LIN {X 0,Y 473.754,Z 554.719,A -85,B 0,C 180,E1 -7288.302,E2 -7288.302} C_VEL
LIN {X 0,Y 473.675,Z 555.595,A -85,B 0,C 180,E1 -7290.002,E2 -7290.002} C_VEL
LIN {X 0,Y 473.755,Z 554.68,A -85,B 0,C 180,E1 -7291.702,E2 -7291.702} C_VEL
LIN {X 0,Y 473.78,Z 553.677,A -85,B 0,C 180,E1 -7292.552,E2 -7292.552} C_VEL
LIN {X 0,Y 473.765,Z 550.247,A -85,B 0,C 180,E1 -7294.255,E2 -7294.255} C_VEL
LIN {X 0,Y 473.855,Z 546.483,A -85,B 0,C 180,E1 -7295.533,E2 -7295.533} C_VEL
LIN {X 0,Y 473.91,Z 541.553,A -85,B 0,C 180,E1 -7296.815,E2 -7296.815} C_VEL
LIN {X 0,Y 474.03,Z 536.5,A -85,B 0,C 180,E1 -7297.883,E2 -7297.883} C_VEL
LIN {X 0,Y 474.244,Z 528.948,A -85,B 0,C 180,E1 -7299.168,E2 -7299.168} C_VEL
LIN {X 0,Y 474.518,Z 521.272,A -85,B 0,C 180,E1 -7300.238,E2 -7300.238} C_VEL
LIN {X 0,Y 474.789,Z 513.997,A -85,B 0,C 180,E1 -7301.095,E2 -7301.095} C_VEL
LIN {X 0,Y 475.091,Z 505.339,A -85,B 0,C 180,E1 -7301.953,E2 -7301.953} C_VEL
LIN {X 0,Y 475.44,Z 496.569,A -85,B 0,C 180,E1 -7302.68,E2 -7302.68} C_VEL
LIN {X 0,Y 475.821,Z 486.805,A -85,B 0,C 180,E1 -7303.344,E2 -7303.344} C_VEL
LIN {X 0,Y 476.16,Z 475.842,A -85,B 0,C 180,E1 -7303.932,E2 -7303.932} C_VEL
LIN {X 0,Y 476.528,Z 464.628,A -85,B 0,C 180,E1 -7304.384,E2 -7304.384} C_VEL
LIN {X 0,Y 476.701,Z 454.582,A -85,B 0,C 180,E1 -7304.679,E2 -7304.679} C_VEL
LIN {X 0,Y 477.021,Z 436.414,A -85,B 0,C 180,E1 -7304.996,E2 -7304.996} C_VEL
LIN {X 0,Y 477.483,Z 358.709,A -85,B 0,C 180,E1 -7306.226,E2 -7306.226} C_VEL
LIN {X 0,Y 475.642,Z 344.411,A -85,B 0,C 180,E1 -7306.547,E2 -7306.547} C_VEL
LIN {X 0,Y 476.419,Z 320.349,A -85,B 0,C 180,E1 -7309.833,E2 -7309.833} C_VEL
LIN {X 0,Y 477.019,Z 300.73,A -85,B 0,C 180,E1 -7312.523,E2 -7312.523} C_VEL
LIN {X 0,Y 477.194,Z 294.12,A -85,B 0,C 180,E1 -7313.431,E2 -7313.431} C_VEL
LIN {X 0,Y 474.603,Z 281.369,A -85,B 0,C 180,E1 -7315.375,E2 -7315.375} C_VEL
LIN {X 0,Y 474.595,Z 281.371,A -85,B 0,C 180,E1 -7318.285,E2 -7318.285} C_VEL
LIN {X 0,Y 474.587,Z 281.373,A -85,B 0,C 180,E1 -7321.217,E2 -7321.217} C_VEL
LIN {X 0,Y 474.622,Z 281.363,A -85,B 0,C 180,E1 -7324.24,E2 -7324.24} C_VEL
LIN {X 0,Y 474.578,Z 281.372,A -85,B 0,C 180,E1 -7327.383,E2 -7327.383} C_VEL
LIN {X 0,Y 474.614,Z 281.369,A -85,B 0,C 180,E1 -7329.646,E2 -7329.646} C_VEL
LIN {X 0,Y 474.62,Z 281.363,A -85,B 0,C 180,E1 -7332.931,E2 -7332.931} C_VEL
LIN {X 0,Y 474.592,Z 281.37,A -85,B 0,C 180,E1 -7335.894,E2 -7335.894} C_VEL
LIN {X 0,Y 474.622,Z 281.361,A -85,B 0,C 180,E1 -7339.038,E2 -7339.038} C_VEL
LIN {X 0,Y 474.597,Z 281.367,A -85,B 0,C 180,E1 -7341.702,E2 -7341.702} C_VEL
LIN {X 0,Y 474.609,Z 281.36,A -85,B 0,C 180,E1 -7344.725,E2 -7344.725} C_VEL
LIN {X 0,Y 474.613,Z 281.358,A -85,B 0,C 180,E1 -7347.787,E2 -7347.787} C_VEL
LIN {X 0,Y 474.605,Z 281.361,A -85,B 0,C 180,E1 -7350.882,E2 -7350.882} C_VEL
LIN {X 0,Y 474.641,Z 281.356,A -85,B 0,C 180,E1 -7353.628,E2 -7353.628} C_VEL
LIN {X 0,Y 474.626,Z 281.365,A -85,B 0,C 180,E1 -7356.635,E2 -7356.635} C_VEL
LIN {X 0,Y 474.647,Z 281.359,A -85,B 0,C 180,E1 -7359.185,E2 -7359.185} C_VEL
LIN {X 0,Y 474.626,Z 281.361,A -85,B 0,C 180,E1 -7361.884,E2 -7361.884} C_VEL
LIN {X 0,Y 474.673,Z 281.359,A -85,B 0,C 180,E1 -7364.544,E2 -7364.544} C_VEL
LIN {X 0,Y 474.708,Z 281.351,A -85,B 0,C 180,E1 -7368.038,E2 -7368.038} C_VEL
LIN {X 0,Y 474.697,Z 281.358,A -85,B 0,C 180,E1 -7371.486,E2 -7371.486} C_VEL
LIN {X 0,Y 474.741,Z 281.351,A -85,B 0,C 180,E1 -7374.052,E2 -7374.052} C_VEL
LIN {X 0,Y 475.065,Z 281.408,A -85,B 0,C 180,E1 -7378.464,E2 -7378.464} C_VEL
LIN {X 0,Y 475.103,Z 295.62,A -85,B 0,C 180,E1 -7380.424,E2 -7380.424} C_VEL
LIN {X 0,Y 474.942,Z 318.084,A -85,B 0,C 180,E1 -7383.606,E2 -7383.606} C_VEL
LIN {X 0,Y 474.942,Z 337.98,A -85,B 0,C 180,E1 -7386.532,E2 -7386.532} C_VEL
LIN {X 0,Y 477.042,Z 351.72,A -85,B 0,C 180,E1 -7386.849,E2 -7386.849} C_VEL
LIN {X 0,Y 476.308,Z 419.465,A -85,B 0,C 180,E1 -7388.038,E2 -7388.038} C_VEL
LIN {X 0,Y 476.073,Z 429.32,A -85,B 0,C 180,E1 -7388.321,E2 -7388.321} C_VEL
LIN {X 0,Y 475.865,Z 440.918,A -85,B 0,C 180,E1 -7388.814,E2 -7388.814} C_VEL
LIN {X 0,Y 475.594,Z 451.584,A -85,B 0,C 180,E1 -7389.463,E2 -7389.463} C_VEL
LIN {X 0,Y 475.26,Z 460.046,A -85,B 0,C 180,E1 -7390.114,E2 -7390.114} C_VEL
LIN {X 0,Y 474.988,Z 468.045,A -85,B 0,C 180,E1 -7390.875,E2 -7390.875} C_VEL
LIN {X 0,Y 474.737,Z 475.533,A -85,B 0,C 180,E1 -7391.745,E2 -7391.745} C_VEL
LIN {X 0,Y 474.418,Z 483.161,A -85,B 0,C 180,E1 -7392.839,E2 -7392.839} C_VEL
LIN {X 0,Y 474.236,Z 489.09,A -85,B 0,C 180,E1 -7393.935,E2 -7393.935} C_VEL
LIN {X 0,Y 474.045,Z 493.784,A -85,B 0,C 180,E1 -7395.038,E2 -7395.038} C_VEL
LIN {X 0,Y 474.004,Z 496.671,A -85,B 0,C 180,E1 -7395.876,E2 -7395.876} C_VEL
LIN {X 0,Y 473.861,Z 499.177,A -85,B 0,C 180,E1 -7396.811,E2 -7396.811} C_VEL
LIN {X 0,Y 473.742,Z 501.689,A -85,B 0,C 180,E1 -7398.308,E2 -7398.308} C_VEL
LIN {X 0,Y 473.721,Z 502.436,A -85,B 0,C 180,E1 -7399.05,E2 -7399.05} C_VEL
LIN {X 0,Y 473.704,Z 502.745,A -85,B 0,C 180,E1 -7399.953,E2 -7399.953} C_VEL
LIN {X 0,Y 473.737,Z 502.436,A -85,B 0,C 180,E1 -7400.858,E2 -7400.858} C_VEL
LIN {X 0,Y 473.745,Z 501.571,A -85,B 0,C 180,E1 -7401.77,E2 -7401.77} C_VEL
LIN {X 0,Y 473.861,Z 499.207,A -85,B 0,C 180,E1 -7403.15,E2 -7403.15} C_VEL
LIN {X 0,Y 473.952,Z 495.309,A -85,B 0,C 180,E1 -7404.532,E2 -7404.532} C_VEL
LIN {X 0,Y 474.097,Z 490.734,A -85,B 0,C 180,E1 -7405.697,E2 -7405.697} C_VEL
LIN {X 0,Y 474.256,Z 486.107,A -85,B 0,C 180,E1 -7406.634,E2 -7406.634} C_VEL
LIN {X 0,Y 474.425,Z 480.407,A -85,B 0,C 180,E1 -7407.577,E2 -7407.577} C_VEL
LIN {X 0,Y 474.636,Z 475.336,A -85,B 0,C 180,E1 -7408.284,E2 -7408.284} C_VEL
LIN {X 0,Y 474.878,Z 467.599,A -85,B 0,C 180,E1 -7409.177,E2 -7409.177} C_VEL
LIN {X 0,Y 475.138,Z 460.809,A -85,B 0,C 180,E1 -7409.826,E2 -7409.826} C_VEL
LIN {X 0,Y 475.404,Z 453.366,A -85,B 0,C 180,E1 -7410.42,E2 -7410.42} C_VEL
LIN {X 0,Y 475.62,Z 445.316,A -85,B 0,C 180,E1 -7410.947,E2 -7410.947} C_VEL
LIN {X 0,Y 475.864,Z 435.766,A -85,B 0,C 180,E1 -7411.435,E2 -7411.435} C_VEL
LIN {X 0,Y 476.027,Z 426.259,A -85,B 0,C 180,E1 -7411.796,E2 -7411.796} C_VEL
LIN {X 0,Y 476.136,Z 415.495,A -85,B 0,C 180,E1 -7412.068,E2 -7412.068} C_VEL
LIN {X 0,Y 476.662,Z 350.671,A -85,B 0,C 180,E1 -7413.144,E2 -7413.144} C_VEL
LIN {X 0,Y 474.823,Z 338.887,A -85,B 0,C 180,E1 -7413.414,E2 -7413.414} C_VEL
LIN {X 0,Y 475.351,Z 320.689,A -85,B 0,C 180,E1 -7416.774,E2 -7416.774} C_VEL
LIN {X 0,Y 475.806,Z 305.452,A -85,B 0,C 180,E1 -7419.63,E2 -7419.63} C_VEL
LIN {X 0,Y 476.229,Z 290.615,A -85,B 0,C 180,E1 -7422.453,E2 -7422.453} C_VEL
LIN {X 0,Y 475.255,Z 284.67,A -85,B 0,C 180,E1 -7423.652,E2 -7423.652} C_VEL
LIN {X 0,Y 474.567,Z 283.121,A -85,B 0,C 180,E1 -7424.071,E2 -7424.071} C_VEL
LIN {X 0,Y 472.887,Z 282.021,A -85,B 0,C 180,E1 -7424.737,E2 -7424.737} C_VEL
LIN {X 0,Y 469.638,Z 281.983,A -85,B 0,C 180,E1 -7425.887,E2 -7425.887} C_VEL
LIN {X 0,Y 467.816,Z 282.217,A -85,B 0,C 180,E1 -7426.852,E2 -7426.852} C_VEL
LIN {X 0,Y 467.568,Z 282.244,A -85,B 0,C 180,E1 -7427.346,E2 -7427.346} C_VEL
LIN {X 0,Y 467.565,Z 282.239,A -85,B 0,C 180,E1 -7430.049,E2 -7430.049} C_VEL
LIN {X 0,Y 467.506,Z 282.246,A -85,B 0,C 180,E1 -7433.038,E2 -7433.038} C_VEL
LIN {X 0,Y 467.563,Z 282.241,A -85,B 0,C 180,E1 -7436.212,E2 -7436.212} C_VEL
LIN {X 0,Y 467.562,Z 282.238,A -85,B 0,C 180,E1 -7439.267,E2 -7439.267} C_VEL
LIN {X 0,Y 467.549,Z 282.243,A -85,B 0,C 180,E1 -7442.483,E2 -7442.483} C_VEL
LIN {X 0,Y 467.559,Z 282.238,A -85,B 0,C 180,E1 -7445.111,E2 -7445.111} C_VEL
LIN {X 0,Y 467.526,Z 282.244,A -85,B 0,C 180,E1 -7447.926,E2 -7447.926} C_VEL
LIN {X 0,Y 467.62,Z 282.239,A -85,B 0,C 180,E1 -7450.692,E2 -7450.692} C_VEL
LIN {X 0,Y 467.641,Z 282.23,A -85,B 0,C 180,E1 -7454.305,E2 -7454.305} C_VEL
LIN {X 0,Y 467.661,Z 282.225,A -85,B 0,C 180,E1 -7457.854,E2 -7457.854} C_VEL
LIN {X 0,Y 467.639,Z 282.236,A -85,B 0,C 180,E1 -7461.356,E2 -7461.356} C_VEL
LIN {X 0,Y 467.706,Z 282.221,A -85,B 0,C 180,E1 -7463.961,E2 -7463.961} C_VEL
LIN {X 0,Y 467.813,Z 282.213,A -85,B 0,C 180,E1 -7467.415,E2 -7467.415} C_VEL
LIN {X 0,Y 467.852,Z 282.207,A -85,B 0,C 180,E1 -7469.998,E2 -7469.998} C_VEL
LIN {X 0,Y 467.813,Z 282.207,A -85,B 0,C 180,E1 -7472.581,E2 -7472.581} C_VEL
LIN {X 0,Y 467.702,Z 282.229,A -85,B 0,C 180,E1 -7476.036,E2 -7476.036} C_VEL
LIN {X 0,Y 467.634,Z 282.232,A -85,B 0,C 180,E1 -7478.641,E2 -7478.641} C_VEL
LIN {X 0,Y 467.655,Z 282.231,A -85,B 0,C 180,E1 -7482.142,E2 -7482.142} C_VEL
LIN {X 0,Y 467.646,Z 282.227,A -85,B 0,C 180,E1 -7485.881,E2 -7485.881} C_VEL
LIN {X 0,Y 467.613,Z 282.234,A -85,B 0,C 180,E1 -7489.304,E2 -7489.304} C_VEL
LIN {X 0,Y 467.522,Z 282.242,A -85,B 0,C 180,E1 -7492.07,E2 -7492.07} C_VEL
LIN {X 0,Y 467.557,Z 282.243,A -85,B 0,C 180,E1 -7494.885,E2 -7494.885} C_VEL
LIN {X 0,Y 467.565,Z 282.24,A -85,B 0,C 180,E1 -7497.768,E2 -7497.768} C_VEL
LIN {X 0,Y 467.55,Z 282.242,A -85,B 0,C 180,E1 -7501.04,E2 -7501.04} C_VEL
LIN {X 0,Y 467.568,Z 282.239,A -85,B 0,C 180,E1 -7504.238,E2 -7504.238} C_VEL
LIN {X 0,Y 467.524,Z 282.243,A -85,B 0,C 180,E1 -7507.182,E2 -7507.182} C_VEL
LIN {X 0,Y 467.548,Z 282.245,A -85,B 0,C 180,E1 -7510.26,E2 -7510.26} C_VEL
LIN {X 0,Y 467.559,Z 282.241,A -85,B 0,C 180,E1 -7512.562,E2 -7512.562} C_VEL
LIN {X 0,Y 467.534,Z 282.242,A -85,B 0,C 180,E1 -7515.048,E2 -7515.048} C_VEL
LIN {X 0,Y 467.556,Z 282.238,A -85,B 0,C 180,E1 -7517.436,E2 -7517.436} C_VEL
LIN {X 0,Y 467.544,Z 282.246,A -85,B 0,C 180,E1 -7520.851,E2 -7520.851} C_VEL
LIN {X 0,Y 467.52,Z 282.244,A -85,B 0,C 180,E1 -7524.257,E2 -7524.257} C_VEL
LIN {X 0,Y 467.53,Z 282.246,A -85,B 0,C 180,E1 -7527.319,E2 -7527.319} C_VEL
LIN {X 0,Y 467.531,Z 282.243,A -85,B 0,C 180,E1 -7530.662,E2 -7530.662} C_VEL
LIN {X 0,Y 467.572,Z 282.243,A -85,B 0,C 180,E1 -7533.196,E2 -7533.196} C_VEL
LIN {X 0,Y 467.543,Z 282.24,A -85,B 0,C 180,E1 -7536.465,E2 -7536.465} C_VEL
LIN {X 0,Y 467.569,Z 282.246,A -85,B 0,C 180,E1 -7539.774,E2 -7539.774} C_VEL
LIN {X 0,Y 467.553,Z 282.24,A -85,B 0,C 180,E1 -7542.504,E2 -7542.504} C_VEL
LIN {X 0,Y 467.553,Z 282.239,A -85,B 0,C 180,E1 -7545.194,E2 -7545.194} C_VEL
LIN {X 0,Y 467.638,Z 282.232,A -85,B 0,C 180,E1 -7547.854,E2 -7547.854} C_VEL
LIN {X 0,Y 467.623,Z 282.23,A -85,B 0,C 180,E1 -7551.356,E2 -7551.356} C_VEL
LIN {X 0,Y 467.694,Z 282.223,A -85,B 0,C 180,E1 -7553.962,E2 -7553.962} C_VEL
LIN {X 0,Y 467.807,Z 282.208,A -85,B 0,C 180,E1 -7557.416,E2 -7557.416} C_VEL
LIN {X 0,Y 467.768,Z 282.22,A -85,B 0,C 180,E1 -7560.86,E2 -7560.86} C_VEL
LIN {X 0,Y 467.806,Z 282.21,A -85,B 0,C 180,E1 -7562.583,E2 -7562.583} C_VEL
LIN {X 0,Y 467.692,Z 282.222,A -85,B 0,C 180,E1 -7566.038,E2 -7566.038} C_VEL
LIN {X 0,Y 467.622,Z 282.231,A -85,B 0,C 180,E1 -7568.643,E2 -7568.643} C_VEL
LIN {X 0,Y 467.631,Z 282.229,A -85,B 0,C 180,E1 -7572.378,E2 -7572.378} C_VEL
LIN {X 0,Y 467.591,Z 282.242,A -85,B 0,C 180,E1 -7575.886,E2 -7575.886} C_VEL
LIN {X 0,Y 467.566,Z 282.238,A -85,B 0,C 180,E1 -7579.31,E2 -7579.31} C_VEL
LIN {X 0,Y 467.496,Z 282.254,A -85,B 0,C 180,E1 -7582.075,E2 -7582.075} C_VEL
LIN {X 0,Y 467.552,Z 282.24,A -85,B 0,C 180,E1 -7584.89,E2 -7584.89} C_VEL
LIN {X 0,Y 467.569,Z 282.237,A -85,B 0,C 180,E1 -7587.772,E2 -7587.772} C_VEL
LIN {X 0,Y 467.517,Z 282.247,A -85,B 0,C 180,E1 -7591.047,E2 -7591.047} C_VEL
LIN {X 0,Y 467.543,Z 282.241,A -85,B 0,C 180,E1 -7594.245,E2 -7594.245} C_VEL
LIN {X 0,Y 467.504,Z 282.251,A -85,B 0,C 180,E1 -7597.19,E2 -7597.19} C_VEL
LIN {X 0,Y 467.529,Z 282.242,A -85,B 0,C 180,E1 -7600.269,E2 -7600.269} C_VEL
LIN {X 0,Y 467.51,Z 282.248,A -85,B 0,C 180,E1 -7603.749,E2 -7603.749} C_VEL
LIN {X 0,Y 467.515,Z 282.244,A -85,B 0,C 180,E1 -7606.259,E2 -7606.259} C_VEL
LIN {X 0,Y 467.545,Z 282.24,A -85,B 0,C 180,E1 -7608.727,E2 -7608.727} C_VEL
LIN {X 0,Y 467.513,Z 282.252,A -85,B 0,C 180,E1 -7611.957,E2 -7611.957} C_VEL
LIN {X 0,Y 467.527,Z 282.242,A -85,B 0,C 180,E1 -7615.17,E2 -7615.17} C_VEL
LIN {X 0,Y 467.551,Z 282.248,A -85,B 0,C 180,E1 -7618.263,E2 -7618.263} C_VEL
LIN {X 0,Y 467.52,Z 282.247,A -85,B 0,C 180,E1 -7621.252,E2 -7621.252} C_VEL
LIN {X 0,Y 467.551,Z 282.367,A -85,B 0,C 180,E1 -7623.832,E2 -7623.832} C_VEL
LIN {X 0,Y 470.766,Z 296.959,A -85,B 0,C 180,E1 -7626.234,E2 -7626.234} C_VEL
LIN {X 0,Y 470.25,Z 310.806,A -85,B 0,C 180,E1 -7628.295,E2 -7628.295} C_VEL
LIN {X 0,Y 469.236,Z 332.306,A -85,B 0,C 180,E1 -7631.445,E2 -7631.445} C_VEL
LIN {X 0,Y 468.72,Z 345.191,A -85,B 0,C 180,E1 -7633.287,E2 -7633.287} C_VEL
LIN {X 0,Y 470.689,Z 361.146,A -85,B 0,C 180,E1 -7633.61,E2 -7633.61} C_VEL
LIN {X 0,Y 469.93,Z 450.761,A -85,B 0,C 180,E1 -7635.053,E2 -7635.053} C_VEL
LIN {X 0,Y 469.719,Z 460.554,A -85,B 0,C 180,E1 -7635.296,E2 -7635.296} C_VEL
LIN {X 0,Y 469.421,Z 470.479,A -85,B 0,C 180,E1 -7635.646,E2 -7635.646} C_VEL
LIN {X 0,Y 469.063,Z 480.775,A -85,B 0,C 180,E1 -7636.133,E2 -7636.133} C_VEL
LIN {X 0,Y 468.663,Z 491.41,A -85,B 0,C 180,E1 -7636.783,E2 -7636.783} C_VEL
LIN {X 0,Y 468.381,Z 500.623,A -85,B 0,C 180,E1 -7637.481,E2 -7637.481} C_VEL
LIN {X 0,Y 468.037,Z 508.608,A -85,B 0,C 180,E1 -7638.197,E2 -7638.197} C_VEL
LIN {X 0,Y 467.648,Z 517.597,A -85,B 0,C 180,E1 -7639.175,E2 -7639.175} C_VEL
LIN {X 0,Y 467.317,Z 525.834,A -85,B 0,C 180,E1 -7640.262,E2 -7640.262} C_VEL
LIN {X 0,Y 467.076,Z 532.675,A -85,B 0,C 180,E1 -7641.349,E2 -7641.349} C_VEL
LIN {X 0,Y 466.926,Z 537.384,A -85,B 0,C 180,E1 -7642.217,E2 -7642.217} C_VEL
LIN {X 0,Y 466.784,Z 543.283,A -85,B 0,C 180,E1 -7643.567,E2 -7643.567} C_VEL
LIN {X 0,Y 466.764,Z 547.601,A -85,B 0,C 180,E1 -7644.819,E2 -7644.819} C_VEL
LIN {X 0,Y 466.666,Z 549.931,A -85,B 0,C 180,E1 -7645.684,E2 -7645.684} C_VEL
LIN {X 0,Y 466.697,Z 553.35,A -85,B 0,C 180,E1 -7647.413,E2 -7647.413} C_VEL
LIN {X 0,Y 466.689,Z 554.318,A -85,B 0,C 180,E1 -7648.276,E2 -7648.276} C_VEL
LIN {X 0,Y 466.604,Z 555.2,A -85,B 0,C 180,E1 -7650.002,E2 -7650.002} C_VEL
LIN {X 0,Y 466.69,Z 554.285,A -85,B 0,C 180,E1 -7651.727,E2 -7651.727} C_VEL
LIN {X 0,Y 466.698,Z 553.276,A -85,B 0,C 180,E1 -7652.591,E2 -7652.591} C_VEL
LIN {X 0,Y 466.673,Z 549.835,A -85,B 0,C 180,E1 -7654.32,E2 -7654.32} C_VEL
LIN {X 0,Y 466.766,Z 546.058,A -85,B 0,C 180,E1 -7655.618,E2 -7655.618} C_VEL
LIN {X 0,Y 466.834,Z 541.109,A -85,B 0,C 180,E1 -7656.918,E2 -7656.918} C_VEL
LIN {X 0,Y 466.98,Z 536.051,A -85,B 0,C 180,E1 -7658.003,E2 -7658.003} C_VEL
LIN {X 0,Y 467.187,Z 528.49,A -85,B 0,C 180,E1 -7659.307,E2 -7659.307} C_VEL
LIN {X 0,Y 467.411,Z 522.541,A -85,B 0,C 180,E1 -7660.177,E2 -7660.177} C_VEL
LIN {X 0,Y 467.795,Z 513.531,A -85,B 0,C 180,E1 -7661.263,E2 -7661.263} C_VEL
LIN {X 0,Y 468.123,Z 504.854,A -85,B 0,C 180,E1 -7662.134,E2 -7662.134} C_VEL
LIN {X 0,Y 468.504,Z 495.716,A -85,B 0,C 180,E1 -7662.895,E2 -7662.895} C_VEL
LIN {X 0,Y 468.894,Z 486.232,A -85,B 0,C 180,E1 -7663.545,E2 -7663.545} C_VEL
LIN {X 0,Y 469.261,Z 475.194,A -85,B 0,C 180,E1 -7664.141,E2 -7664.141} C_VEL
LIN {X 0,Y 469.611,Z 464.686,A -85,B 0,C 180,E1 -7664.573,E2 -7664.573} C_VEL
LIN {X 0,Y 469.82,Z 453.545,A -85,B 0,C 180,E1 -7664.899,E2 -7664.899} C_VEL
LIN {X 0,Y 470.155,Z 433.395,A -85,B 0,C 180,E1 -7665.248,E2 -7665.248} C_VEL
LIN {X 0,Y 470.607,Z 359.16,A -85,B 0,C 180,E1 -7666.45,E2 -7666.45} C_VEL
LIN {X 0,Y 468.696,Z 344.431,A -85,B 0,C 180,E1 -7666.783,E2 -7666.783} C_VEL
LIN {X 0,Y 469.499,Z 321.988,A -85,B 0,C 180,E1 -7669.887,E2 -7669.887} C_VEL
LIN {X 0,Y 470.149,Z 302.171,A -85,B 0,C 180,E1 -7672.638,E2 -7672.638} C_VEL
LIN {X 0,Y 470.314,Z 295.607,A -85,B 0,C 180,E1 -7673.561,E2 -7673.561} C_VEL
LIN {X 0,Y 467.565,Z 282.246,A -85,B 0,C 180,E1 -7675.628,E2 -7675.628} C_VEL
LIN {X 0,Y 467.535,Z 282.252,A -85,B 0,C 180,E1 -7678.751,E2 -7678.751} C_VEL
LIN {X 0,Y 467.572,Z 282.245,A -85,B 0,C 180,E1 -7681.739,E2 -7681.739} C_VEL
LIN {X 0,Y 467.554,Z 282.243,A -85,B 0,C 180,E1 -7684.832,E2 -7684.832} C_VEL
LIN {X 0,Y 467.553,Z 282.247,A -85,B 0,C 180,E1 -7688.043,E2 -7688.043} C_VEL
LIN {X 0,Y 467.568,Z 282.244,A -85,B 0,C 180,E1 -7691.276,E2 -7691.276} C_VEL
LIN {X 0,Y 467.551,Z 282.247,A -85,B 0,C 180,E1 -7693.821,E2 -7693.821} C_VEL
LIN {X 0,Y 467.539,Z 282.247,A -85,B 0,C 180,E1 -7696.254,E2 -7696.254} C_VEL
LIN {X 0,Y 467.566,Z 282.24,A -85,B 0,C 180,E1 -7698.721,E2 -7698.721} C_VEL
LIN {X 0,Y 467.555,Z 282.242,A -85,B 0,C 180,E1 -7701.406,E2 -7701.406} C_VEL
LIN {X 0,Y 467.543,Z 282.244,A -85,B 0,C 180,E1 -7704.259,E2 -7704.259} C_VEL
LIN {X 0,Y 467.559,Z 282.234,A -85,B 0,C 180,E1 -7707.32,E2 -7707.32} C_VEL
LIN {X 0,Y 467.552,Z 282.242,A -85,B 0,C 180,E1 -7710.665,E2 -7710.665} C_VEL
LIN {X 0,Y 467.594,Z 282.234,A -85,B 0,C 180,E1 -7713.199,E2 -7713.199} C_VEL
LIN {X 0,Y 467.563,Z 282.242,A -85,B 0,C 180,E1 -7716.057,E2 -7716.057} C_VEL
LIN {X 0,Y 467.613,Z 282.239,A -85,B 0,C 180,E1 -7718.857,E2 -7718.857} C_VEL
LIN {X 0,Y 467.602,Z 282.236,A -85,B 0,C 180,E1 -7721.602,E2 -7721.602} C_VEL
LIN {X 0,Y 467.611,Z 282.238,A -85,B 0,C 180,E1 -7724.304,E2 -7724.304} C_VEL
LIN {X 0,Y 467.667,Z 282.228,A -85,B 0,C 180,E1 -7727.855,E2 -7727.855} C_VEL
LIN {X 0,Y 467.651,Z 282.236,A -85,B 0,C 180,E1 -7731.357,E2 -7731.357} C_VEL
LIN {X 0,Y 467.705,Z 282.228,A -85,B 0,C 180,E1 -7733.963,E2 -7733.963} C_VEL
LIN {X 0,Y 468.038,Z 282.309,A -85,B 0,C 180,E1 -7738.28,E2 -7738.28} C_VEL
LIN {X 0,Y 468.287,Z 286.877,A -85,B 0,C 180,E1 -7738.926,E2 -7738.926} C_VEL
LIN {X 0,Y 468.051,Z 306.795,A -85,B 0,C 180,E1 -7741.721,E2 -7741.721} C_VEL
LIN {X 0,Y 467.943,Z 327.588,A -85,B 0,C 180,E1 -7744.739,E2 -7744.739} C_VEL
LIN {X 0,Y 467.971,Z 338.082,A -85,B 0,C 180,E1 -7746.278,E2 -7746.278} C_VEL
LIN {X 0,Y 470.189,Z 352.34,A -85,B 0,C 180,E1 -7746.626,E2 -7746.626} C_VEL
LIN {X 0,Y 469.417,Z 419.947,A -85,B 0,C 180,E1 -7747.844,E2 -7747.844} C_VEL
LIN {X 0,Y 469.176,Z 430.173,A -85,B 0,C 180,E1 -7748.146,E2 -7748.146} C_VEL
LIN {X 0,Y 468.951,Z 441.053,A -85,B 0,C 180,E1 -7748.62,E2 -7748.62} C_VEL
LIN {X 0,Y 468.666,Z 451.771,A -85,B 0,C 180,E1 -7749.277,E2 -7749.277} C_VEL
LIN {X 0,Y 468.332,Z 460.253,A -85,B 0,C 180,E1 -7749.938,E2 -7749.938} C_VEL
LIN {X 0,Y 468.041,Z 467.26,A -85,B 0,C 180,E1 -7750.6,E2 -7750.6} C_VEL
LIN {X 0,Y 467.801,Z 473.212,A -85,B 0,C 180,E1 -7751.263,E2 -7751.263} C_VEL
LIN {X 0,Y 467.554,Z 479.825,A -85,B 0,C 180,E1 -7752.149,E2 -7752.149} C_VEL
LIN {X 0,Y 467.327,Z 485.336,A -85,B 0,C 180,E1 -7753.038,E2 -7753.038} C_VEL
LIN {X 0,Y 467.168,Z 489.922,A -85,B 0,C 180,E1 -7753.928,E2 -7753.928} C_VEL
LIN {X 0,Y 466.96,Z 495.1,A -85,B 0,C 180,E1 -7755.211,E2 -7755.211} C_VEL
LIN {X 0,Y 466.867,Z 498.056,A -85,B 0,C 180,E1 -7756.171,E2 -7756.171} C_VEL
LIN {X 0,Y 466.807,Z 499.265,A -85,B 0,C 180,E1 -7756.622,E2 -7756.622} C_VEL
LIN {X 0,Y 466.724,Z 501.047,A -85,B 0,C 180,E1 -7757.528,E2 -7757.528} C_VEL
LIN {X 0,Y 466.648,Z 502.271,A -85,B 0,C 180,E1 -7758.438,E2 -7758.438} C_VEL
LIN {X 0,Y 466.625,Z 502.948,A -85,B 0,C 180,E1 -7759.351,E2 -7759.351} C_VEL
LIN {X 0,Y 466.626,Z 503.083,A -85,B 0,C 180,E1 -7760.268,E2 -7760.268} C_VEL
LIN {X 0,Y 466.65,Z 502.651,A -85,B 0,C 180,E1 -7761.19,E2 -7761.19} C_VEL
LIN {X 0,Y 466.699,Z 501.574,A -85,B 0,C 180,E1 -7762.116,E2 -7762.116} C_VEL
LIN {X 0,Y 466.791,Z 499.329,A -85,B 0,C 180,E1 -7763.314,E2 -7763.314} C_VEL
LIN {X 0,Y 466.899,Z 496.174,A -85,B 0,C 180,E1 -7764.453,E2 -7764.453} C_VEL
LIN {X 0,Y 466.993,Z 492.517,A -85,B 0,C 180,E1 -7765.457,E2 -7765.457} C_VEL
LIN {X 0,Y 467.178,Z 487.223,A -85,B 0,C 180,E1 -7766.587,E2 -7766.587} C_VEL
LIN {X 0,Y 467.369,Z 482.073,A -85,B 0,C 180,E1 -7767.483,E2 -7767.483} C_VEL
LIN {X 0,Y 467.629,Z 474.861,A -85,B 0,C 180,E1 -7768.501,E2 -7768.501} C_VEL
LIN {X 0,Y 467.901,Z 467.725,A -85,B 0,C 180,E1 -7769.327,E2 -7769.327} C_VEL
LIN {X 0,Y 468.171,Z 459.954,A -85,B 0,C 180,E1 -7770.068,E2 -7770.068} C_VEL
LIN {X 0,Y 468.475,Z 450.89,A -85,B 0,C 180,E1 -7770.769,E2 -7770.769} C_VEL
LIN {X 0,Y 468.864,Z 439.171,A -85,B 0,C 180,E1 -7771.458,E2 -7771.458} C_VEL
LIN {X 0,Y 469.052,Z 429.057,A -85,B 0,C 180,E1 -7771.882,E2 -7771.882} C_VEL
LIN {X 0,Y 469.198,Z 419.003,A -85,B 0,C 180,E1 -7772.172,E2 -7772.172} C_VEL
LIN {X 0,Y 469.76,Z 351.311,A -85,B 0,C 180,E1 -7773.338,E2 -7773.338} C_VEL
LIN {X 0,Y 467.828,Z 338.929,A -85,B 0,C 180,E1 -7773.625,E2 -7773.625} C_VEL
LIN {X 0,Y 468.462,Z 319.047,A -85,B 0,C 180,E1 -7777.338,E2 -7777.338} C_VEL
LIN {X 0,Y 468.96,Z 302.932,A -85,B 0,C 180,E1 -7780.403,E2 -7780.403} C_VEL
LIN {X 0,Y 469.237,Z 291.179,A -85,B 0,C 180,E1 -7782.675,E2 -7782.675} C_VEL
LIN {X 0,Y 467.575,Z 282.244,A -85,B 0,C 180,E1 -7784.539,E2 -7784.539} C_VEL
LIN {X 0,Y 467.568,Z 282.244,A -85,B 0,C 180,E1 -7787.346,E2 -7787.346} C_VEL
LIN {X 0,Y 466.946,Z 282.327,A -85,B 0,C 180,E1 -7788.066,E2 -7788.066} C_VEL
LIN {X 0,Y 464.06,Z 282.682,A -85,B 0,C 180,E1 -7789.233,E2 -7789.233} C_VEL
LIN {X 0,Y 461.601,Z 282.982,A -85,B 0,C 180,E1 -7790.175,E2 -7790.175} C_VEL
LIN {X 0,Y 460.566,Z 283.111,A -85,B 0,C 180,E1 -7790.904,E2 -7790.904} C_VEL
LIN {X 0,Y 460.495,Z 283.122,A -85,B 0,C 180,E1 -7791.15,E2 -7791.15} C_VEL
LIN {X 0,Y 460.5,Z 283.117,A -85,B 0,C 180,E1 -7794.555,E2 -7794.555} C_VEL
LIN {X 0,Y 460.522,Z 283.121,A -85,B 0,C 180,E1 -7797.716,E2 -7797.716} C_VEL
LIN {X 0,Y 460.518,Z 283.116,A -85,B 0,C 180,E1 -7800.769,E2 -7800.769} C_VEL
LIN {X 0,Y 460.535,Z 283.122,A -85,B 0,C 180,E1 -7804.208,E2 -7804.208} C_VEL
LIN {X 0,Y 460.498,Z 283.118,A -85,B 0,C 180,E1 -7807.571,E2 -7807.571} C_VEL
LIN {X 0,Y 460.565,Z 283.115,A -85,B 0,C 180,E1 -7810.384,E2 -7810.384} C_VEL
LIN {X 0,Y 460.557,Z 283.114,A -85,B 0,C 180,E1 -7813.146,E2 -7813.146} C_VEL
LIN {X 0,Y 460.544,Z 283.112,A -85,B 0,C 180,E1 -7815.867,E2 -7815.867} C_VEL
LIN {X 0,Y 460.611,Z 283.106,A -85,B 0,C 180,E1 -7818.559,E2 -7818.559} C_VEL
LIN {X 0,Y 460.628,Z 283.102,A -85,B 0,C 180,E1 -7822.106,E2 -7822.106} C_VEL
LIN {X 0,Y 460.677,Z 283.096,A -85,B 0,C 180,E1 -7824.747,E2 -7824.747} C_VEL
LIN {X 0,Y 460.757,Z 283.091,A -85,B 0,C 180,E1 -7827.376,E2 -7827.376} C_VEL
LIN {X 0,Y 460.822,Z 283.082,A -85,B 0,C 180,E1 -7829.998,E2 -7829.998} C_VEL
LIN {X 0,Y 460.757,Z 283.086,A -85,B 0,C 180,E1 -7832.621,E2 -7832.621} C_VEL
LIN {X 0,Y 460.668,Z 283.105,A -85,B 0,C 180,E1 -7836.128,E2 -7836.128} C_VEL
LIN {X 0,Y 460.59,Z 283.108,A -85,B 0,C 180,E1 -7838.774,E2 -7838.774} C_VEL
LIN {X 0,Y 460.608,Z 283.111,A -85,B 0,C 180,E1 -7842.331,E2 -7842.331} C_VEL
LIN {X 0,Y 460.598,Z 283.106,A -85,B 0,C 180,E1 -7845.994,E2 -7845.994} C_VEL
LIN {X 0,Y 460.559,Z 283.11,A -85,B 0,C 180,E1 -7849.612,E2 -7849.612} C_VEL
LIN {X 0,Y 460.498,Z 283.119,A -85,B 0,C 180,E1 -7852.425,E2 -7852.425} C_VEL
LIN {X 0,Y 460.524,Z 283.116,A -85,B 0,C 180,E1 -7855.789,E2 -7855.789} C_VEL
LIN {X 0,Y 460.511,Z 283.116,A -85,B 0,C 180,E1 -7858.231,E2 -7858.231} C_VEL
LIN {X 0,Y 460.503,Z 283.122,A -85,B 0,C 180,E1 -7861.278,E2 -7861.278} C_VEL
LIN {X 0,Y 460.511,Z 283.116,A -85,B 0,C 180,E1 -7864.501,E2 -7864.501} C_VEL
LIN {X 0,Y 460.478,Z 283.125,A -85,B 0,C 180,E1 -7867.619,E2 -7867.619} C_VEL
LIN {X 0,Y 460.513,Z 283.121,A -85,B 0,C 180,E1 -7870.264,E2 -7870.264} C_VEL
LIN {X 0,Y 460.467,Z 283.122,A -85,B 0,C 180,E1 -7873.371,E2 -7873.371} C_VEL
LIN {X 0,Y 460.466,Z 283.127,A -85,B 0,C 180,E1 -7876.62,E2 -7876.62} C_VEL
LIN {X 0,Y 460.506,Z 283.117,A -85,B 0,C 180,E1 -7879.726,E2 -7879.726} C_VEL
LIN {X 0,Y 460.461,Z 283.128,A -85,B 0,C 180,E1 -7882.52,E2 -7882.52} C_VEL
LIN {X 0,Y 460.496,Z 283.119,A -85,B 0,C 180,E1 -7885.619,E2 -7885.619} C_VEL
LIN {X 0,Y 460.494,Z 283.122,A -85,B 0,C 180,E1 -7888.741,E2 -7888.741} C_VEL
LIN {X 0,Y 460.542,Z 283.112,A -85,B 0,C 180,E1 -7892.249,E2 -7892.249} C_VEL
LIN {X 0,Y 460.511,Z 283.116,A -85,B 0,C 180,E1 -7894.702,E2 -7894.702} C_VEL
LIN {X 0,Y 460.464,Z 283.131,A -85,B 0,C 180,E1 -7897.568,E2 -7897.568} C_VEL
LIN {X 0,Y 460.515,Z 283.117,A -85,B 0,C 180,E1 -7900.382,E2 -7900.382} C_VEL
LIN {X 0,Y 460.51,Z 283.116,A -85,B 0,C 180,E1 -7903.144,E2 -7903.144} C_VEL
LIN {X 0,Y 460.505,Z 283.123,A -85,B 0,C 180,E1 -7905.866,E2 -7905.866} C_VEL
LIN {X 0,Y 460.574,Z 283.112,A -85,B 0,C 180,E1 -7908.558,E2 -7908.558} C_VEL
LIN {X 0,Y 460.637,Z 283.104,A -85,B 0,C 180,E1 -7912.107,E2 -7912.107} C_VEL
LIN {X 0,Y 460.646,Z 283.106,A -85,B 0,C 180,E1 -7914.747,E2 -7914.747} C_VEL
LIN {X 0,Y 460.773,Z 283.084,A -85,B 0,C 180,E1 -7917.377,E2 -7917.377} C_VEL
LIN {X 0,Y 460.789,Z 283.081,A -85,B 0,C 180,E1 -7920,E2 -7920} C_VEL
LIN {X 0,Y 460.771,Z 283.087,A -85,B 0,C 180,E1 -7922.622,E2 -7922.622} C_VEL
LIN {X 0,Y 460.657,Z 283.098,A -85,B 0,C 180,E1 -7926.13,E2 -7926.13} C_VEL
LIN {X 0,Y 460.569,Z 283.11,A -85,B 0,C 180,E1 -7928.777,E2 -7928.777} C_VEL
LIN {X 0,Y 460.577,Z 283.108,A -85,B 0,C 180,E1 -7932.458,E2 -7932.458} C_VEL
LIN {X 0,Y 460.544,Z 283.118,A -85,B 0,C 180,E1 -7935.999,E2 -7935.999} C_VEL
LIN {X 0,Y 460.513,Z 283.116,A -85,B 0,C 180,E1 -7938.903,E2 -7938.903} C_VEL
LIN {X 0,Y 460.481,Z 283.121,A -85,B 0,C 180,E1 -7941.487,E2 -7941.487} C_VEL
LIN {X 0,Y 460.492,Z 283.127,A -85,B 0,C 180,E1 -7944.335,E2 -7944.335} C_VEL
LIN {X 0,Y 460.521,Z 283.115,A -85,B 0,C 180,E1 -7947.247,E2 -7947.247} C_VEL
LIN {X 0,Y 460.46,Z 283.126,A -85,B 0,C 180,E1 -7950.243,E2 -7950.243} C_VEL
LIN {X 0,Y 460.482,Z 283.122,A -85,B 0,C 180,E1 -7953.328,E2 -7953.328} C_VEL
LIN {X 0,Y 460.433,Z 283.128,A -85,B 0,C 180,E1 -7956.533,E2 -7956.533} C_VEL
LIN {X 0,Y 460.479,Z 283.121,A -85,B 0,C 180,E1 -7959.867,E2 -7959.867} C_VEL
LIN {X 0,Y 460.454,Z 283.126,A -85,B 0,C 180,E1 -7962.901,E2 -7962.901} C_VEL
LIN {X 0,Y 460.471,Z 283.125,A -85,B 0,C 180,E1 -7965.835,E2 -7965.835} C_VEL
LIN {X 0,Y 460.497,Z 283.118,A -85,B 0,C 180,E1 -7968.992,E2 -7968.992} C_VEL
LIN {X 0,Y 460.456,Z 283.125,A -85,B 0,C 180,E1 -7972.379,E2 -7972.379} C_VEL
LIN {X 0,Y 460.508,Z 283.119,A -85,B 0,C 180,E1 -7975.627,E2 -7975.627} C_VEL
LIN {X 0,Y 460.481,Z 283.123,A -85,B 0,C 180,E1 -7978.746,E2 -7978.746} C_VEL
LIN {X 0,Y 460.484,Z 283.124,A -85,B 0,C 180,E1 -7981.768,E2 -7981.768} C_VEL
LIN {X 0,Y 460.525,Z 283.212,A -85,B 0,C 180,E1 -7983.585,E2 -7983.585} C_VEL
LIN {X 0,Y 463.794,Z 298.215,A -85,B 0,C 180,E1 -7986.091,E2 -7986.091} C_VEL
LIN {X 0,Y 463.804,Z 302.841,A -85,B 0,C 180,E1 -7986.802,E2 -7986.802} C_VEL
LIN {X 0,Y 462.69,Z 324.668,A -85,B 0,C 180,E1 -7990.066,E2 -7990.066} C_VEL
LIN {X 0,Y 461.752,Z 344.979,A -85,B 0,C 180,E1 -7993.06,E2 -7993.06} C_VEL
LIN {X 0,Y 463.805,Z 361.77,A -85,B 0,C 180,E1 -7993.408,E2 -7993.408} C_VEL
LIN {X 0,Y 462.973,Z 451.028,A -85,B 0,C 180,E1 -7994.879,E2 -7994.879} C_VEL
LIN {X 0,Y 462.777,Z 460.631,A -85,B 0,C 180,E1 -7995.126,E2 -7995.126} C_VEL
LIN {X 0,Y 462.456,Z 470.454,A -85,B 0,C 180,E1 -7995.481,E2 -7995.481} C_VEL
LIN {X 0,Y 462.155,Z 479.755,A -85,B 0,C 180,E1 -7995.921,E2 -7995.921} C_VEL
LIN {X 0,Y 461.717,Z 490.54,A -85,B 0,C 180,E1 -7996.581,E2 -7996.581} C_VEL
LIN {X 0,Y 461.395,Z 499.782,A -85,B 0,C 180,E1 -7997.281,E2 -7997.281} C_VEL
LIN {X 0,Y 460.985,Z 508.966,A -85,B 0,C 180,E1 -7998.126,E2 -7998.126} C_VEL
LIN {X 0,Y 460.597,Z 516.989,A -85,B 0,C 180,E1 -7999.007,E2 -7999.007} C_VEL
LIN {X 0,Y 460.274,Z 525.282,A -85,B 0,C 180,E1 -8000.112,E2 -8000.112} C_VEL
LIN {X 0,Y 459.993,Z 532.164,A -85,B 0,C 180,E1 -8001.214,E2 -8001.214} C_VEL
LIN {X 0,Y 459.863,Z 536.896,A -85,B 0,C 180,E1 -8002.097,E2 -8002.097} C_VEL
LIN {X 0,Y 459.707,Z 543.199,A -85,B 0,C 180,E1 -8003.571,E2 -8003.571} C_VEL
LIN {X 0,Y 459.672,Z 547.172,A -85,B 0,C 180,E1 -8004.739,E2 -8004.739} C_VEL
LIN {X 0,Y 459.581,Z 549.504,A -85,B 0,C 180,E1 -8005.617,E2 -8005.617} C_VEL
LIN {X 0,Y 459.617,Z 552.946,A -85,B 0,C 180,E1 -8007.373,E2 -8007.373} C_VEL
LIN {X 0,Y 459.626,Z 553.916,A -85,B 0,C 180,E1 -8008.249,E2 -8008.249} C_VEL
LIN {X 0,Y 459.535,Z 554.804,A -85,B 0,C 180,E1 -8010.002,E2 -8010.002} C_VEL
LIN {X 0,Y 459.61,Z 553.889,A -85,B 0,C 180,E1 -8011.754,E2 -8011.754} C_VEL
LIN {X 0,Y 459.618,Z 552.879,A -85,B 0,C 180,E1 -8012.631,E2 -8012.631} C_VEL
LIN {X 0,Y 459.587,Z 549.436,A -85,B 0,C 180,E1 -8014.386,E2 -8014.386} C_VEL
LIN {X 0,Y 459.661,Z 545.657,A -85,B 0,C 180,E1 -8015.705,E2 -8015.705} C_VEL
LIN {X 0,Y 459.742,Z 540.71,A -85,B 0,C 180,E1 -8017.026,E2 -8017.026} C_VEL
LIN {X 0,Y 459.907,Z 535.643,A -85,B 0,C 180,E1 -8018.127,E2 -8018.127} C_VEL
LIN {X 0,Y 460.087,Z 529.514,A -85,B 0,C 180,E1 -8019.23,E2 -8019.23} C_VEL
LIN {X 0,Y 460.381,Z 522.103,A -85,B 0,C 180,E1 -8020.334,E2 -8020.334} C_VEL
LIN {X 0,Y 460.8,Z 513.073,A -85,B 0,C 180,E1 -8021.437,E2 -8021.437} C_VEL
LIN {X 0,Y 461.153,Z 504.368,A -85,B 0,C 180,E1 -8022.32,E2 -8022.32} C_VEL
LIN {X 0,Y 461.566,Z 494.72,A -85,B 0,C 180,E1 -8023.127,E2 -8023.127} C_VEL
LIN {X 0,Y 461.943,Z 485.656,A -85,B 0,C 180,E1 -8023.752,E2 -8023.752} C_VEL
LIN {X 0,Y 462.323,Z 475.762,A -85,B 0,C 180,E1 -8024.302,E2 -8024.302} C_VEL
LIN {X 0,Y 462.728,Z 463.913,A -85,B 0,C 180,E1 -8024.795,E2 -8024.795} C_VEL
LIN {X 0,Y 462.936,Z 453.838,A -85,B 0,C 180,E1 -8025.097,E2 -8025.097} C_VEL
LIN {X 0,Y 463.288,Z 434.122,A -85,B 0,C 180,E1 -8025.452,E2 -8025.452} C_VEL
LIN {X 0,Y 463.825,Z 360.181,A -85,B 0,C 180,E1 -8026.676,E2 -8026.676} C_VEL
LIN {X 0,Y 461.76,Z 344.323,A -85,B 0,C 180,E1 -8027.043,E2 -8027.043} C_VEL
LIN {X 0,Y 462.565,Z 323.598,A -85,B 0,C 180,E1 -8029.943,E2 -8029.943} C_VEL
LIN {X 0,Y 463.282,Z 303.709,A -85,B 0,C 180,E1 -8032.757,E2 -8032.757} C_VEL
LIN {X 0,Y 463.424,Z 297.09,A -85,B 0,C 180,E1 -8033.695,E2 -8033.695} C_VEL
LIN {X 0,Y 461.02,Z 285.327,A -85,B 0,C 180,E1 -8035.525,E2 -8035.525} C_VEL
LIN {X 0,Y 460.524,Z 283.123,A -85,B 0,C 180,E1 -8035.913,E2 -8035.913} C_VEL
LIN {X 0,Y 460.511,Z 283.129,A -85,B 0,C 180,E1 -8039.232,E2 -8039.232} C_VEL
LIN {X 0,Y 460.522,Z 283.12,A -85,B 0,C 180,E1 -8042.284,E2 -8042.284} C_VEL
LIN {X 0,Y 460.5,Z 283.126,A -85,B 0,C 180,E1 -8045.445,E2 -8045.445} C_VEL
LIN {X 0,Y 460.532,Z 283.119,A -85,B 0,C 180,E1 -8048.896,E2 -8048.896} C_VEL
LIN {X 0,Y 460.51,Z 283.124,A -85,B 0,C 180,E1 -8052.18,E2 -8052.18} C_VEL
LIN {X 0,Y 460.5,Z 283.124,A -85,B 0,C 180,E1 -8055.41,E2 -8055.41} C_VEL
LIN {X 0,Y 460.517,Z 283.121,A -85,B 0,C 180,E1 -8058.396,E2 -8058.396} C_VEL
LIN {X 0,Y 460.52,Z 283.117,A -85,B 0,C 180,E1 -8061.267,E2 -8061.267} C_VEL
LIN {X 0,Y 460.493,Z 283.119,A -85,B 0,C 180,E1 -8064.553,E2 -8064.553} C_VEL
LIN {X 0,Y 460.509,Z 283.114,A -85,B 0,C 180,E1 -8067.714,E2 -8067.714} C_VEL
LIN {X 0,Y 460.521,Z 283.116,A -85,B 0,C 180,E1 -8070.768,E2 -8070.768} C_VEL
LIN {X 0,Y 460.543,Z 283.113,A -85,B 0,C 180,E1 -8073.734,E2 -8073.734} C_VEL
LIN {X 0,Y 460.534,Z 283.12,A -85,B 0,C 180,E1 -8076.624,E2 -8076.624} C_VEL
LIN {X 0,Y 460.544,Z 283.115,A -85,B 0,C 180,E1 -8079.453,E2 -8079.453} C_VEL
LIN {X 0,Y 460.529,Z 283.12,A -85,B 0,C 180,E1 -8082.229,E2 -8082.229} C_VEL
LIN {X 0,Y 460.541,Z 283.121,A -85,B 0,C 180,E1 -8084.965,E2 -8084.965} C_VEL
LIN {X 0,Y 460.628,Z 283.105,A -85,B 0,C 180,E1 -8087.667,E2 -8087.667} C_VEL
LIN {X 0,Y 460.599,Z 283.116,A -85,B 0,C 180,E1 -8091.224,E2 -8091.224} C_VEL
LIN {X 0,Y 460.671,Z 283.104,A -85,B 0,C 180,E1 -8093.87,E2 -8093.87} C_VEL
LIN {X 0,Y 460.928,Z 283.118,A -85,B 0,C 180,E1 -8098.062,E2 -8098.062} C_VEL
LIN {X 0,Y 461.431,Z 287.462,A -85,B 0,C 180,E1 -8098.691,E2 -8098.691} C_VEL
LIN {X 0,Y 461.135,Z 309.003,A -85,B 0,C 180,E1 -8101.747,E2 -8101.747} C_VEL
LIN {X 0,Y 460.973,Z 329.882,A -85,B 0,C 180,E1 -8104.811,E2 -8104.811} C_VEL
LIN {X 0,Y 460.965,Z 337.759,A -85,B 0,C 180,E1 -8105.99,E2 -8105.99} C_VEL
LIN {X 0,Y 463.401,Z 353.549,A -85,B 0,C 180,E1 -8106.395,E2 -8106.395} C_VEL
LIN {X 0,Y 462.519,Z 420.498,A -85,B 0,C 180,E1 -8107.641,E2 -8107.641} C_VEL
LIN {X 0,Y 462.301,Z 431.214,A -85,B 0,C 180,E1 -8107.971,E2 -8107.971} C_VEL
LIN {X 0,Y 461.94,Z 443.769,A -85,B 0,C 180,E1 -8108.565,E2 -8108.565} C_VEL
LIN {X 0,Y 461.661,Z 453.489,A -85,B 0,C 180,E1 -8109.198,E2 -8109.198} C_VEL
LIN {X 0,Y 461.343,Z 461.721,A -85,B 0,C 180,E1 -8109.869,E2 -8109.869} C_VEL
LIN {X 0,Y 461.008,Z 469.588,A -85,B 0,C 180,E1 -8110.653,E2 -8110.653} C_VEL
LIN {X 0,Y 460.681,Z 477.834,A -85,B 0,C 180,E1 -8111.662,E2 -8111.662} C_VEL
LIN {X 0,Y 460.341,Z 484.808,A -85,B 0,C 180,E1 -8112.745,E2 -8112.745} C_VEL
LIN {X 0,Y 460.128,Z 489.771,A -85,B 0,C 180,E1 -8113.695,E2 -8113.695} C_VEL
LIN {X 0,Y 459.981,Z 493.683,A -85,B 0,C 180,E1 -8114.602,E2 -8114.602} C_VEL
LIN {X 0,Y 459.842,Z 498.119,A -85,B 0,C 180,E1 -8115.969,E2 -8115.969} C_VEL
LIN {X 0,Y 459.692,Z 500.372,A -85,B 0,C 180,E1 -8116.887,E2 -8116.887} C_VEL
LIN {X 0,Y 459.62,Z 502.024,A -85,B 0,C 180,E1 -8117.808,E2 -8117.808} C_VEL
LIN {X 0,Y 459.573,Z 503.034,A -85,B 0,C 180,E1 -8118.732,E2 -8118.732} C_VEL
LIN {X 0,Y 459.534,Z 503.462,A -85,B 0,C 180,E1 -8119.662,E2 -8119.662} C_VEL
LIN {X 0,Y 459.568,Z 503.099,A -85,B 0,C 180,E1 -8121.127,E2 -8121.127} C_VEL
LIN {X 0,Y 459.625,Z 501.413,A -85,B 0,C 180,E1 -8122.475,E2 -8122.475} C_VEL
LIN {X 0,Y 459.716,Z 499.39,A -85,B 0,C 180,E1 -8123.48,E2 -8123.48} C_VEL
LIN {X 0,Y 459.819,Z 496.954,A -85,B 0,C 180,E1 -8124.374,E2 -8124.374} C_VEL
LIN {X 0,Y 459.942,Z 492.337,A -85,B 0,C 180,E1 -8125.648,E2 -8125.648} C_VEL
LIN {X 0,Y 460.14,Z 486.974,A -85,B 0,C 180,E1 -8126.781,E2 -8126.781} C_VEL
LIN {X 0,Y 460.352,Z 481.638,A -85,B 0,C 180,E1 -8127.699,E2 -8127.699} C_VEL
LIN {X 0,Y 460.55,Z 476.232,A -85,B 0,C 180,E1 -8128.482,E2 -8128.482} C_VEL
LIN {X 0,Y 460.861,Z 468.895,A -85,B 0,C 180,E1 -8129.361,E2 -8129.361} C_VEL
LIN {X 0,Y 461.135,Z 462.174,A -85,B 0,C 180,E1 -8130.034,E2 -8130.034} C_VEL
LIN {X 0,Y 461.43,Z 454.413,A -85,B 0,C 180,E1 -8130.68,E2 -8130.68} C_VEL
LIN {X 0,Y 461.663,Z 446.144,A -85,B 0,C 180,E1 -8131.242,E2 -8131.242} C_VEL
LIN {X 0,Y 461.944,Z 436.972,A -85,B 0,C 180,E1 -8131.731,E2 -8131.731} C_VEL
LIN {X 0,Y 462.116,Z 427.318,A -85,B 0,C 180,E1 -8132.116,E2 -8132.116} C_VEL
LIN {X 0,Y 462.249,Z 417.112,A -85,B 0,C 180,E1 -8132.392,E2 -8132.392} C_VEL
LIN {X 0,Y 462.845,Z 351.918,A -85,B 0,C 180,E1 -8133.536,E2 -8133.536} C_VEL
LIN {X 0,Y 460.829,Z 338.984,A -85,B 0,C 180,E1 -8133.836,E2 -8133.836} C_VEL
LIN {X 0,Y 461.424,Z 320.847,A -85,B 0,C 180,E1 -8137.261,E2 -8137.261} C_VEL
LIN {X 0,Y 462.001,Z 304.062,A -85,B 0,C 180,E1 -8140.487,E2 -8140.487} C_VEL
LIN {X 0,Y 462.326,Z 293.396,A -85,B 0,C 180,E1 -8142.568,E2 -8142.568} C_VEL
LIN {X 0,Y 460.969,Z 285.375,A -85,B 0,C 180,E1 -8144.232,E2 -8144.232} C_VEL
LIN {X 0,Y 460.538,Z 283.121,A -85,B 0,C 180,E1 -8144.719,E2 -8144.719} C_VEL
LIN {X 0,Y 460.523,Z 283.116,A -85,B 0,C 180,E1 -8148.4,E2 -8148.4} C_VEL
LIN {X 0,Y 460.495,Z 283.122,A -85,B 0,C 180,E1 -8151.15,E2 -8151.15} C_VEL
LIN {X 0,Y 459.861,Z 283.206,A -85,B 0,C 180,E1 -8151.881,E2 -8151.881} C_VEL
LIN {X 0,Y 457.009,Z 283.559,A -85,B 0,C 180,E1 -8153.067,E2 -8153.067} C_VEL
LIN {X 0,Y 454.583,Z 283.858,A -85,B 0,C 180,E1 -8154.023,E2 -8154.023} C_VEL
LIN {X 0,Y 453.549,Z 283.983,A -85,B 0,C 180,E1 -8154.762,E2 -8154.762} C_VEL
LIN {X 0,Y 453.47,Z 283.994,A -85,B 0,C 180,E1 -8155.013,E2 -8155.013} C_VEL
LIN {X 0,Y 453.458,Z 283.999,A -85,B 0,C 180,E1 -8158.202,E2 -8158.202} C_VEL
LIN {X 0,Y 453.461,Z 283.995,A -85,B 0,C 180,E1 -8161.286,E2 -8161.286} C_VEL
LIN {X 0,Y 453.493,Z 283.999,A -85,B 0,C 180,E1 -8164.284,E2 -8164.284} C_VEL
LIN {X 0,Y 453.465,Z 283.994,A -85,B 0,C 180,E1 -8167.204,E2 -8167.204} C_VEL
LIN {X 0,Y 453.499,Z 283.992,A -85,B 0,C 180,E1 -8170.066,E2 -8170.066} C_VEL
LIN {X 0,Y 453.498,Z 283.997,A -85,B 0,C 180,E1 -8172.875,E2 -8172.875} C_VEL
LIN {X 0,Y 453.505,Z 283.989,A -85,B 0,C 180,E1 -8175.643,E2 -8175.643} C_VEL
LIN {X 0,Y 453.561,Z 283.983,A -85,B 0,C 180,E1 -8178.378,E2 -8178.378} C_VEL
LIN {X 0,Y 453.565,Z 283.988,A -85,B 0,C 180,E1 -8181.085,E2 -8181.085} C_VEL
LIN {X 0,Y 453.64,Z 283.975,A -85,B 0,C 180,E1 -8183.773,E2 -8183.773} C_VEL
LIN {X 0,Y 453.704,Z 283.969,A -85,B 0,C 180,E1 -8187.335,E2 -8187.335} C_VEL
LIN {X 0,Y 453.771,Z 283.961,A -85,B 0,C 180,E1 -8189.998,E2 -8189.998} C_VEL
LIN {X 0,Y 453.704,Z 283.964,A -85,B 0,C 180,E1 -8192.661,E2 -8192.661} C_VEL
LIN {X 0,Y 453.636,Z 283.979,A -85,B 0,C 180,E1 -8196.223,E2 -8196.223} C_VEL
LIN {X 0,Y 453.56,Z 283.983,A -85,B 0,C 180,E1 -8198.911,E2 -8198.911} C_VEL
LIN {X 0,Y 453.563,Z 283.99,A -85,B 0,C 180,E1 -8202.526,E2 -8202.526} C_VEL
LIN {X 0,Y 453.541,Z 283.987,A -85,B 0,C 180,E1 -8206.193,E2 -8206.193} C_VEL
LIN {X 0,Y 453.511,Z 283.994,A -85,B 0,C 180,E1 -8209.035,E2 -8209.035} C_VEL
LIN {X 0,Y 453.468,Z 283.993,A -85,B 0,C 180,E1 -8211.832,E2 -8211.832} C_VEL
LIN {X 0,Y 453.479,Z 283.995,A -85,B 0,C 180,E1 -8214.732,E2 -8214.732} C_VEL
LIN {X 0,Y 453.476,Z 283.994,A -85,B 0,C 180,E1 -8217.945,E2 -8217.945} C_VEL
LIN {X 0,Y 453.459,Z 283.995,A -85,B 0,C 180,E1 -8220.755,E2 -8220.755} C_VEL
LIN {X 0,Y 453.457,Z 284,A -85,B 0,C 180,E1 -8223.908,E2 -8223.908} C_VEL
LIN {X 0,Y 453.429,Z 283.999,A -85,B 0,C 180,E1 -8227.185,E2 -8227.185} C_VEL
LIN {X 0,Y 453.468,Z 283.995,A -85,B 0,C 180,E1 -8230.604,E2 -8230.604} C_VEL
LIN {X 0,Y 453.431,Z 284.007,A -85,B 0,C 180,E1 -8234.217,E2 -8234.217} C_VEL
LIN {X 0,Y 453.43,Z 284,A -85,B 0,C 180,E1 -8237,E2 -8237} C_VEL
LIN {X 0,Y 453.468,Z 284.001,A -85,B 0,C 180,E1 -8240.547,E2 -8240.547} C_VEL
LIN {X 0,Y 453.415,Z 284,A -85,B 0,C 180,E1 -8243.913,E2 -8243.913} C_VEL
LIN {X 0,Y 453.431,Z 284.005,A -85,B 0,C 180,E1 -8247.146,E2 -8247.146} C_VEL
LIN {X 0,Y 453.47,Z 283.993,A -85,B 0,C 180,E1 -8250.267,E2 -8250.267} C_VEL
LIN {X 0,Y 453.463,Z 284.002,A -85,B 0,C 180,E1 -8253.291,E2 -8253.291} C_VEL
LIN {X 0,Y 453.454,Z 283.996,A -85,B 0,C 180,E1 -8256.236,E2 -8256.236} C_VEL
LIN {X 0,Y 453.431,Z 284,A -85,B 0,C 180,E1 -8259.115,E2 -8259.115} C_VEL
LIN {X 0,Y 453.457,Z 284.003,A -85,B 0,C 180,E1 -8261.942,E2 -8261.942} C_VEL
LIN {X 0,Y 453.485,Z 283.992,A -85,B 0,C 180,E1 -8264.724,E2 -8264.724} C_VEL
LIN {X 0,Y 453.547,Z 283.984,A -85,B 0,C 180,E1 -8267.47,E2 -8267.47} C_VEL
LIN {X 0,Y 453.534,Z 283.986,A -85,B 0,C 180,E1 -8271.085,E2 -8271.085} C_VEL
LIN {X 0,Y 453.624,Z 283.974,A -85,B 0,C 180,E1 -8273.773,E2 -8273.773} C_VEL
LIN {X 0,Y 453.714,Z 283.964,A -85,B 0,C 180,E1 -8277.336,E2 -8277.336} C_VEL
LIN {X 0,Y 453.76,Z 283.957,A -85,B 0,C 180,E1 -8280,E2 -8280} C_VEL
LIN {X 0,Y 453.713,Z 283.966,A -85,B 0,C 180,E1 -8282.663,E2 -8282.663} C_VEL
LIN {X 0,Y 453.623,Z 283.974,A -85,B 0,C 180,E1 -8286.226,E2 -8286.226} C_VEL
LIN {X 0,Y 453.533,Z 283.988,A -85,B 0,C 180,E1 -8288.914,E2 -8288.914} C_VEL
LIN {X 0,Y 453.545,Z 283.984,A -85,B 0,C 180,E1 -8292.552,E2 -8292.552} C_VEL
LIN {X 0,Y 453.489,Z 283.994,A -85,B 0,C 180,E1 -8296.197,E2 -8296.197} C_VEL
LIN {X 0,Y 453.463,Z 283.994,A -85,B 0,C 180,E1 -8299.041,E2 -8299.041} C_VEL
LIN {X 0,Y 453.434,Z 284.002,A -85,B 0,C 180,E1 -8301.838,E2 -8301.838} C_VEL
LIN {X 0,Y 453.463,Z 283.997,A -85,B 0,C 180,E1 -8304.737,E2 -8304.737} C_VEL
LIN {X 0,Y 453.481,Z 283.994,A -85,B 0,C 180,E1 -8307.962,E2 -8307.962} C_VEL
LIN {X 0,Y 453.417,Z 284,A -85,B 0,C 180,E1 -8311.528,E2 -8311.528} C_VEL
LIN {X 0,Y 453.443,Z 284.004,A -85,B 0,C 180,E1 -8314.781,E2 -8314.781} C_VEL
LIN {X 0,Y 453.419,Z 284,A -85,B 0,C 180,E1 -8318.316,E2 -8318.316} C_VEL
LIN {X 0,Y 453.454,Z 283.996,A -85,B 0,C 180,E1 -8320.613,E2 -8320.613} C_VEL
LIN {X 0,Y 453.422,Z 283.999,A -85,B 0,C 180,E1 -8324.226,E2 -8324.226} C_VEL
LIN {X 0,Y 453.427,Z 284,A -85,B 0,C 180,E1 -8327.009,E2 -8327.009} C_VEL
LIN {X 0,Y 453.463,Z 283.999,A -85,B 0,C 180,E1 -8329.413,E2 -8329.413} C_VEL
LIN {X 0,Y 453.41,Z 284.001,A -85,B 0,C 180,E1 -8332.813,E2 -8332.813} C_VEL
LIN {X 0,Y 453.44,Z 284.006,A -85,B 0,C 180,E1 -8336.09,E2 -8336.09} C_VEL
LIN {X 0,Y 453.433,Z 283.999,A -85,B 0,C 180,E1 -8339.243,E2 -8339.243} C_VEL
LIN {X 0,Y 453.452,Z 284.004,A -85,B 0,C 180,E1 -8342.297,E2 -8342.297} C_VEL
LIN {X 0,Y 453.468,Z 284.142,A -85,B 0,C 180,E1 -8343.343,E2 -8343.343} C_VEL
LIN {X 0,Y 456.853,Z 299.451,A -85,B 0,C 180,E1 -8345.946,E2 -8345.946} C_VEL
LIN {X 0,Y 456.898,Z 304.077,A -85,B 0,C 180,E1 -8346.671,E2 -8346.671} C_VEL
LIN {X 0,Y 455.751,Z 325.597,A -85,B 0,C 180,E1 -8349.938,E2 -8349.938} C_VEL
LIN {X 0,Y 454.783,Z 345.181,A -85,B 0,C 180,E1 -8352.842,E2 -8352.842} C_VEL
LIN {X 0,Y 456.91,Z 361.702,A -85,B 0,C 180,E1 -8353.195,E2 -8353.195} C_VEL
LIN {X 0,Y 456.068,Z 450.013,A -85,B 0,C 180,E1 -8354.673,E2 -8354.673} C_VEL
LIN {X 0,Y 455.856,Z 459.874,A -85,B 0,C 180,E1 -8354.924,E2 -8354.924} C_VEL
LIN {X 0,Y 455.509,Z 470.432,A -85,B 0,C 180,E1 -8355.312,E2 -8355.312} C_VEL
LIN {X 0,Y 455.138,Z 480.608,A -85,B 0,C 180,E1 -8355.814,E2 -8355.814} C_VEL
LIN {X 0,Y 454.686,Z 491.167,A -85,B 0,C 180,E1 -8356.483,E2 -8356.483} C_VEL
LIN {X 0,Y 454.373,Z 500.074,A -85,B 0,C 180,E1 -8357.179,E2 -8357.179} C_VEL
LIN {X 0,Y 453.933,Z 509.293,A -85,B 0,C 180,E1 -8358.052,E2 -8358.052} C_VEL
LIN {X 0,Y 453.514,Z 518.071,A -85,B 0,C 180,E1 -8359.06,E2 -8359.06} C_VEL
LIN {X 0,Y 453.209,Z 524.688,A -85,B 0,C 180,E1 -8359.956,E2 -8359.956} C_VEL
LIN {X 0,Y 452.943,Z 531.615,A -85,B 0,C 180,E1 -8361.076,E2 -8361.076} C_VEL
LIN {X 0,Y 452.812,Z 536.363,A -85,B 0,C 180,E1 -8361.973,E2 -8361.973} C_VEL
LIN {X 0,Y 452.638,Z 542.334,A -85,B 0,C 180,E1 -8363.36,E2 -8363.36} C_VEL
LIN {X 0,Y 452.582,Z 546.714,A -85,B 0,C 180,E1 -8364.656,E2 -8364.656} C_VEL
LIN {X 0,Y 452.501,Z 549.048,A -85,B 0,C 180,E1 -8365.548,E2 -8365.548} C_VEL
LIN {X 0,Y 452.539,Z 552.526,A -85,B 0,C 180,E1 -8367.332,E2 -8367.332} C_VEL
LIN {X 0,Y 452.488,Z 554.115,A -85,B 0,C 180,E1 -8369.112,E2 -8369.112} C_VEL
LIN {X 0,Y 452.468,Z 554.404,A -85,B 0,C 180,E1 -8370.002,E2 -8370.002} C_VEL
LIN {X 0,Y 452.52,Z 553.501,A -85,B 0,C 180,E1 -8371.782,E2 -8371.782} C_VEL
LIN {X 0,Y 452.54,Z 552.488,A -85,B 0,C 180,E1 -8372.672,E2 -8372.672} C_VEL
LIN {X 0,Y 452.507,Z 549.05,A -85,B 0,C 180,E1 -8374.455,E2 -8374.455} C_VEL
LIN {X 0,Y 452.558,Z 545.266,A -85,B 0,C 180,E1 -8375.795,E2 -8375.795} C_VEL
LIN {X 0,Y 452.667,Z 540.313,A -85,B 0,C 180,E1 -8377.136,E2 -8377.136} C_VEL
LIN {X 0,Y 452.829,Z 535.235,A -85,B 0,C 180,E1 -8378.255,E2 -8378.255} C_VEL
LIN {X 0,Y 453.024,Z 529.092,A -85,B 0,C 180,E1 -8379.376,E2 -8379.376} C_VEL
LIN {X 0,Y 453.352,Z 521.666,A -85,B 0,C 180,E1 -8380.496,E2 -8380.496} C_VEL
LIN {X 0,Y 453.805,Z 512.611,A -85,B 0,C 180,E1 -8381.615,E2 -8381.615} C_VEL
LIN {X 0,Y 454.179,Z 503.901,A -85,B 0,C 180,E1 -8382.512,E2 -8382.512} C_VEL
LIN {X 0,Y 454.605,Z 494.544,A -85,B 0,C 180,E1 -8383.31,E2 -8383.31} C_VEL
LIN {X 0,Y 455.008,Z 485.191,A -85,B 0,C 180,E1 -8383.966,E2 -8383.966} C_VEL
LIN {X 0,Y 455.415,Z 475.296,A -85,B 0,C 180,E1 -8384.524,E2 -8384.524} C_VEL
LIN {X 0,Y 455.869,Z 463.448,A -85,B 0,C 180,E1 -8385.022,E2 -8385.022} C_VEL
LIN {X 0,Y 456.083,Z 453.328,A -85,B 0,C 180,E1 -8385.33,E2 -8385.33} C_VEL
LIN {X 0,Y 456.421,Z 435.28,A -85,B 0,C 180,E1 -8385.661,E2 -8385.661} C_VEL
LIN {X 0,Y 457.026,Z 360.87,A -85,B 0,C 180,E1 -8386.919,E2 -8386.919} C_VEL
LIN {X 0,Y 454.845,Z 344.288,A -85,B 0,C 180,E1 -8387.31,E2 -8387.31} C_VEL
LIN {X 0,Y 455.702,Z 323.253,A -85,B 0,C 180,E1 -8390.304,E2 -8390.304} C_VEL
LIN {X 0,Y 456.493,Z 303.547,A -85,B 0,C 180,E1 -8393.115,E2 -8393.115} C_VEL
LIN {X 0,Y 456.572,Z 298.744,A -85,B 0,C 180,E1 -8393.813,E2 -8393.813} C_VEL
LIN {X 0,Y 453.893,Z 285.78,A -85,B 0,C 180,E1 -8395.873,E2 -8395.873} C_VEL
LIN {X 0,Y 453.478,Z 284,A -85,B 0,C 180,E1 -8396.2,E2 -8396.2} C_VEL
LIN {X 0,Y 453.454,Z 284.007,A -85,B 0,C 180,E1 -8398.715,E2 -8398.715} C_VEL
LIN {X 0,Y 453.455,Z 284.004,A -85,B 0,C 180,E1 -8401.799,E2 -8401.799} C_VEL
LIN {X 0,Y 453.47,Z 283.999,A -85,B 0,C 180,E1 -8404.988,E2 -8404.988} C_VEL
LIN {X 0,Y 453.452,Z 284.002,A -85,B 0,C 180,E1 -8408.311,E2 -8408.311} C_VEL
LIN {X 0,Y 453.482,Z 283.997,A -85,B 0,C 180,E1 -8410.608,E2 -8410.608} C_VEL
LIN {X 0,Y 453.448,Z 284.002,A -85,B 0,C 180,E1 -8413.244,E2 -8413.244} C_VEL
LIN {X 0,Y 453.449,Z 284.003,A -85,B 0,C 180,E1 -8415.778,E2 -8415.778} C_VEL
LIN {X 0,Y 453.499,Z 283.994,A -85,B 0,C 180,E1 -8419.404,E2 -8419.404} C_VEL
LIN {X 0,Y 453.457,Z 283.999,A -85,B 0,C 180,E1 -8422.222,E2 -8422.222} C_VEL
LIN {X 0,Y 453.468,Z 283.991,A -85,B 0,C 180,E1 -8425.221,E2 -8425.221} C_VEL
LIN {X 0,Y 453.444,Z 283.999,A -85,B 0,C 180,E1 -8428.474,E2 -8428.474} C_VEL
LIN {X 0,Y 453.49,Z 283.989,A -85,B 0,C 180,E1 -8431.287,E2 -8431.287} C_VEL
LIN {X 0,Y 453.516,Z 283.992,A -85,B 0,C 180,E1 -8434.285,E2 -8434.285} C_VEL
LIN {X 0,Y 453.474,Z 283.997,A -85,B 0,C 180,E1 -8437.204,E2 -8437.204} C_VEL
LIN {X 0,Y 453.483,Z 283.997,A -85,B 0,C 180,E1 -8440.066,E2 -8440.066} C_VEL
LIN {X 0,Y 453.477,Z 284,A -85,B 0,C 180,E1 -8442.875,E2 -8442.875} C_VEL
LIN {X 0,Y 453.492,Z 283.993,A -85,B 0,C 180,E1 -8445.644,E2 -8445.644} C_VEL
LIN {X 0,Y 453.558,Z 283.988,A -85,B 0,C 180,E1 -8448.379,E2 -8448.379} C_VEL
LIN {X 0,Y 453.621,Z 283.982,A -85,B 0,C 180,E1 -8451.985,E2 -8451.985} C_VEL
LIN {X 0,Y 453.636,Z 283.984,A -85,B 0,C 180,E1 -8454.667,E2 -8454.667} C_VEL
LIN {X 0,Y 453.862,Z 284.07,A -85,B 0,C 180,E1 -8457.837,E2 -8457.837} C_VEL
LIN {X 0,Y 454.557,Z 288.119,A -85,B 0,C 180,E1 -8458.45,E2 -8458.45} C_VEL
LIN {X 0,Y 454.224,Z 309.749,A -85,B 0,C 180,E1 -8461.552,E2 -8461.552} C_VEL
LIN {X 0,Y 454.048,Z 330.784,A -85,B 0,C 180,E1 -8464.662,E2 -8464.662} C_VEL
LIN {X 0,Y 454.014,Z 337.813,A -85,B 0,C 180,E1 -8465.72,E2 -8465.72} C_VEL
LIN {X 0,Y 456.631,Z 354.593,A -85,B 0,C 180,E1 -8466.158,E2 -8466.158} C_VEL
LIN {X 0,Y 455.656,Z 420.965,A -85,B 0,C 180,E1 -8467.422,E2 -8467.422} C_VEL
LIN {X 0,Y 455.437,Z 431.646,A -85,B 0,C 180,E1 -8467.761,E2 -8467.761} C_VEL
LIN {X 0,Y 455.073,Z 443.761,A -85,B 0,C 180,E1 -8468.34,E2 -8468.34} C_VEL
LIN {X 0,Y 454.755,Z 453.806,A -85,B 0,C 180,E1 -8469.003,E2 -8469.003} C_VEL
LIN {X 0,Y 454.399,Z 462.036,A -85,B 0,C 180,E1 -8469.684,E2 -8469.684} C_VEL
LIN {X 0,Y 454.044,Z 469.897,A -85,B 0,C 180,E1 -8470.479,E2 -8470.479} C_VEL
LIN {X 0,Y 453.655,Z 478.959,A -85,B 0,C 180,E1 -8471.619,E2 -8471.619} C_VEL
LIN {X 0,Y 453.292,Z 485.98,A -85,B 0,C 180,E1 -8472.765,E2 -8472.765} C_VEL
LIN {X 0,Y 453.063,Z 490.605,A -85,B 0,C 180,E1 -8473.684,E2 -8473.684} C_VEL
LIN {X 0,Y 452.892,Z 495.229,A -85,B 0,C 180,E1 -8474.836,E2 -8474.836} C_VEL
LIN {X 0,Y 452.742,Z 499.393,A -85,B 0,C 180,E1 -8476.226,E2 -8476.226} C_VEL
LIN {X 0,Y 452.584,Z 501.387,A -85,B 0,C 180,E1 -8477.161,E2 -8477.161} C_VEL
LIN {X 0,Y 452.488,Z 503.408,A -85,B 0,C 180,E1 -8478.669,E2 -8478.669} C_VEL
LIN {X 0,Y 452.467,Z 503.953,A -85,B 0,C 180,E1 -8479.982,E2 -8479.982} C_VEL
LIN {X 0,Y 452.5,Z 503.359,A -85,B 0,C 180,E1 -8481.279,E2 -8481.279} C_VEL
LIN {X 0,Y 452.571,Z 501.141,A -85,B 0,C 180,E1 -8482.845,E2 -8482.845} C_VEL
LIN {X 0,Y 452.738,Z 497.691,A -85,B 0,C 180,E1 -8484.291,E2 -8484.291} C_VEL
LIN {X 0,Y 452.891,Z 492.542,A -85,B 0,C 180,E1 -8485.754,E2 -8485.754} C_VEL
LIN {X 0,Y 453.073,Z 488.048,A -85,B 0,C 180,E1 -8486.734,E2 -8486.734} C_VEL
LIN {X 0,Y 453.304,Z 482.512,A -85,B 0,C 180,E1 -8487.718,E2 -8487.718} C_VEL
LIN {X 0,Y 453.561,Z 475.69,A -85,B 0,C 180,E1 -8488.709,E2 -8488.709} C_VEL
LIN {X 0,Y 453.889,Z 468.418,A -85,B 0,C 180,E1 -8489.575,E2 -8489.575} C_VEL
LIN {X 0,Y 454.194,Z 460.678,A -85,B 0,C 180,E1 -8490.335,E2 -8490.335} C_VEL
LIN {X 0,Y 454.524,Z 451.469,A -85,B 0,C 180,E1 -8491.069,E2 -8491.069} C_VEL
LIN {X 0,Y 454.945,Z 440.533,A -85,B 0,C 180,E1 -8491.742,E2 -8491.742} C_VEL
LIN {X 0,Y 455.159,Z 429.091,A -85,B 0,C 180,E1 -8492.236,E2 -8492.236} C_VEL
LIN {X 0,Y 455.315,Z 419.787,A -85,B 0,C 180,E1 -8492.513,E2 -8492.513} C_VEL
LIN {X 0,Y 456.002,Z 353.128,A -85,B 0,C 180,E1 -8493.718,E2 -8493.718} C_VEL
LIN {X 0,Y 453.835,Z 338.993,A -85,B 0,C 180,E1 -8494.06,E2 -8494.06} C_VEL
LIN {X 0,Y 454.507,Z 320.222,A -85,B 0,C 180,E1 -8497.647,E2 -8497.647} C_VEL
LIN {X 0,Y 455.08,Z 303.902,A -85,B 0,C 180,E1 -8500.827,E2 -8500.827} C_VEL
LIN {X 0,Y 455.349,Z 294.055,A -85,B 0,C 180,E1 -8502.775,E2 -8502.775} C_VEL
LIN {X 0,Y 453.512,Z 283.996,A -85,B 0,C 180,E1 -8504.92,E2 -8504.92} C_VEL
LIN {X 0,Y 453.47,Z 283.995,A -85,B 0,C 180,E1 -8508.211,E2 -8508.211} C_VEL
LIN {X 0,Y 453.429,Z 284,A -85,B 0,C 180,E1 -8511.149,E2 -8511.149} C_VEL
LIN {X 0,Y 453.442,Z 284.002,A -85,B 0,C 180,E1 -8513.918,E2 -8513.918} C_VEL
LIN {X 0,Y 453.47,Z 283.994,A -85,B 0,C 180,E1 -8515.013,E2 -8515.013} C_VEL
LIN {X 0,Y 452.817,Z 284.084,A -85,B 0,C 180,E1 -8515.754,E2 -8515.754} C_VEL
LIN {X 0,Y 449.963,Z 284.434,A -85,B 0,C 180,E1 -8516.958,E2 -8516.958} C_VEL
LIN {X 0,Y 447.534,Z 284.741,A -85,B 0,C 180,E1 -8517.929,E2 -8517.929} C_VEL
LIN {X 0,Y 446.485,Z 284.864,A -85,B 0,C 180,E1 -8518.68,E2 -8518.68} C_VEL
LIN {X 0,Y 446.396,Z 284.874,A -85,B 0,C 180,E1 -8518.934,E2 -8518.934} C_VEL
LIN {X 0,Y 446.423,Z 284.876,A -85,B 0,C 180,E1 -8521.837,E2 -8521.837} C_VEL
LIN {X 0,Y 446.421,Z 284.873,A -85,B 0,C 180,E1 -8524.846,E2 -8524.846} C_VEL
LIN {X 0,Y 446.448,Z 284.873,A -85,B 0,C 180,E1 -8528.247,E2 -8528.247} C_VEL
LIN {X 0,Y 446.452,Z 284.867,A -85,B 0,C 180,E1 -8531.649,E2 -8531.649} C_VEL
LIN {X 0,Y 446.48,Z 284.868,A -85,B 0,C 180,E1 -8534.478,E2 -8534.478} C_VEL
LIN {X 0,Y 446.52,Z 284.859,A -85,B 0,C 180,E1 -8538.192,E2 -8538.192} C_VEL
LIN {X 0,Y 446.516,Z 284.864,A -85,B 0,C 180,E1 -8540.943,E2 -8540.943} C_VEL
LIN {X 0,Y 446.61,Z 284.852,A -85,B 0,C 180,E1 -8543.675,E2 -8543.675} C_VEL
LIN {X 0,Y 446.653,Z 284.847,A -85,B 0,C 180,E1 -8547.293,E2 -8547.293} C_VEL
LIN {X 0,Y 446.721,Z 284.839,A -85,B 0,C 180,E1 -8549.998,E2 -8549.998} C_VEL
LIN {X 0,Y 446.653,Z 284.842,A -85,B 0,C 180,E1 -8552.704,E2 -8552.704} C_VEL
LIN {X 0,Y 446.606,Z 284.854,A -85,B 0,C 180,E1 -8556.322,E2 -8556.322} C_VEL
LIN {X 0,Y 446.511,Z 284.86,A -85,B 0,C 180,E1 -8559.053,E2 -8559.053} C_VEL
LIN {X 0,Y 446.521,Z 284.864,A -85,B 0,C 180,E1 -8562.727,E2 -8562.727} C_VEL
LIN {X 0,Y 446.485,Z 284.869,A -85,B 0,C 180,E1 -8566.456,E2 -8566.456} C_VEL
LIN {X 0,Y 446.462,Z 284.869,A -85,B 0,C 180,E1 -8569.3,E2 -8569.3} C_VEL
LIN {X 0,Y 446.408,Z 284.873,A -85,B 0,C 180,E1 -8572.196,E2 -8572.196} C_VEL
LIN {X 0,Y 446.421,Z 284.88,A -85,B 0,C 180,E1 -8575.15,E2 -8575.15} C_VEL
LIN {X 0,Y 446.427,Z 284.871,A -85,B 0,C 180,E1 -8578.177,E2 -8578.177} C_VEL
LIN {X 0,Y 446.399,Z 284.879,A -85,B 0,C 180,E1 -8581.296,E2 -8581.296} C_VEL
LIN {X 0,Y 446.409,Z 284.873,A -85,B 0,C 180,E1 -8584.519,E2 -8584.519} C_VEL
LIN {X 0,Y 446.389,Z 284.882,A -85,B 0,C 180,E1 -8588.074,E2 -8588.074} C_VEL
LIN {X 0,Y 446.399,Z 284.874,A -85,B 0,C 180,E1 -8590.913,E2 -8590.913} C_VEL
LIN {X 0,Y 446.368,Z 284.881,A -85,B 0,C 180,E1 -8593.842,E2 -8593.842} C_VEL
LIN {X 0,Y 446.366,Z 284.887,A -85,B 0,C 180,E1 -8596.399,E2 -8596.399} C_VEL
LIN {X 0,Y 446.393,Z 284.877,A -85,B 0,C 180,E1 -8599.078,E2 -8599.078} C_VEL
LIN {X 0,Y 446.377,Z 284.877,A -85,B 0,C 180,E1 -8601.917,E2 -8601.917} C_VEL
LIN {X 0,Y 446.382,Z 284.878,A -85,B 0,C 180,E1 -8605.472,E2 -8605.472} C_VEL
LIN {X 0,Y 446.372,Z 284.881,A -85,B 0,C 180,E1 -8608.696,E2 -8608.696} C_VEL
LIN {X 0,Y 446.44,Z 284.871,A -85,B 0,C 180,E1 -8611.818,E2 -8611.818} C_VEL
LIN {X 0,Y 446.409,Z 284.874,A -85,B 0,C 180,E1 -8614.844,E2 -8614.844} C_VEL
LIN {X 0,Y 446.398,Z 284.875,A -85,B 0,C 180,E1 -8618.242,E2 -8618.242} C_VEL
LIN {X 0,Y 446.403,Z 284.879,A -85,B 0,C 180,E1 -8621.646,E2 -8621.646} C_VEL
LIN {X 0,Y 446.453,Z 284.87,A -85,B 0,C 180,E1 -8624.477,E2 -8624.477} C_VEL
LIN {X 0,Y 446.488,Z 284.872,A -85,B 0,C 180,E1 -8628.192,E2 -8628.192} C_VEL
LIN {X 0,Y 446.543,Z 284.858,A -85,B 0,C 180,E1 -8631.856,E2 -8631.856} C_VEL
LIN {X 0,Y 446.593,Z 284.859,A -85,B 0,C 180,E1 -8634.581,E2 -8634.581} C_VEL
LIN {X 0,Y 446.659,Z 284.843,A -85,B 0,C 180,E1 -8637.294,E2 -8637.294} C_VEL
LIN {X 0,Y 446.731,Z 284.833,A -85,B 0,C 180,E1 -8640,E2 -8640} C_VEL
LIN {X 0,Y 446.657,Z 284.846,A -85,B 0,C 180,E1 -8642.705,E2 -8642.705} C_VEL
LIN {X 0,Y 446.591,Z 284.85,A -85,B 0,C 180,E1 -8646.324,E2 -8646.324} C_VEL
LIN {X 0,Y 446.479,Z 284.868,A -85,B 0,C 180,E1 -8649.056,E2 -8649.056} C_VEL
LIN {X 0,Y 446.478,Z 284.864,A -85,B 0,C 180,E1 -8652.73,E2 -8652.73} C_VEL
LIN {X 0,Y 446.434,Z 284.871,A -85,B 0,C 180,E1 -8656.461,E2 -8656.461} C_VEL
LIN {X 0,Y 446.415,Z 284.873,A -85,B 0,C 180,E1 -8659.305,E2 -8659.305} C_VEL
LIN {X 0,Y 446.375,Z 284.886,A -85,B 0,C 180,E1 -8662.201,E2 -8662.201} C_VEL
LIN {X 0,Y 446.406,Z 284.873,A -85,B 0,C 180,E1 -8665.155,E2 -8665.155} C_VEL
LIN {X 0,Y 446.436,Z 284.873,A -85,B 0,C 180,E1 -8668.181,E2 -8668.181} C_VEL
LIN {X 0,Y 446.37,Z 284.877,A -85,B 0,C 180,E1 -8671.777,E2 -8671.777} C_VEL
LIN {X 0,Y 446.384,Z 284.88,A -85,B 0,C 180,E1 -8674.526,E2 -8674.526} C_VEL
LIN {X 0,Y 446.371,Z 284.877,A -85,B 0,C 180,E1 -8678.082,E2 -8678.082} C_VEL
LIN {X 0,Y 446.383,Z 284.88,A -85,B 0,C 180,E1 -8680.92,E2 -8680.92} C_VEL
LIN {X 0,Y 446.36,Z 284.882,A -85,B 0,C 180,E1 -8683.85,E2 -8683.85} C_VEL
LIN {X 0,Y 446.361,Z 284.879,A -85,B 0,C 180,E1 -8686.408,E2 -8686.408} C_VEL
LIN {X 0,Y 446.395,Z 284.876,A -85,B 0,C 180,E1 -8689.087,E2 -8689.087} C_VEL
LIN {X 0,Y 446.364,Z 284.884,A -85,B 0,C 180,E1 -8692.123,E2 -8692.123} C_VEL
LIN {X 0,Y 446.394,Z 284.876,A -85,B 0,C 180,E1 -8695.48,E2 -8695.48} C_VEL
LIN {X 0,Y 446.385,Z 284.88,A -85,B 0,C 180,E1 -8698.703,E2 -8698.703} C_VEL
LIN {X 0,Y 446.403,Z 284.879,A -85,B 0,C 180,E1 -8701.84,E2 -8701.84} C_VEL
LIN {X 0,Y 446.398,Z 284.896,A -85,B 0,C 180,E1 -8703.069,E2 -8703.069} C_VEL
LIN {X 0,Y 449.92,Z 300.843,A -85,B 0,C 180,E1 -8705.827,E2 -8705.827} C_VEL
LIN {X 0,Y 450.001,Z 305.287,A -85,B 0,C 180,E1 -8706.536,E2 -8706.536} C_VEL
LIN {X 0,Y 448.709,Z 327.826,A -85,B 0,C 180,E1 -8710.01,E2 -8710.01} C_VEL
LIN {X 0,Y 447.809,Z 344.999,A -85,B 0,C 180,E1 -8712.611,E2 -8712.611} C_VEL
LIN {X 0,Y 450.023,Z 363.072,A -85,B 0,C 180,E1 -8713.001,E2 -8713.001} C_VEL
LIN {X 0,Y 449.123,Z 450.262,A -85,B 0,C 180,E1 -8714.489,E2 -8714.489} C_VEL
LIN {X 0,Y 448.898,Z 459.94,A -85,B 0,C 180,E1 -8714.742,E2 -8714.742} C_VEL
LIN {X 0,Y 448.558,Z 470.405,A -85,B 0,C 180,E1 -8715.137,E2 -8715.137} C_VEL
LIN {X 0,Y 448.201,Z 479.58,A -85,B 0,C 180,E1 -8715.589,E2 -8715.589} C_VEL
LIN {X 0,Y 447.736,Z 490.281,A -85,B 0,C 180,E1 -8716.269,E2 -8716.269} C_VEL
LIN {X 0,Y 447.356,Z 500.345,A -85,B 0,C 180,E1 -8717.072,E2 -8717.072} C_VEL
LIN {X 0,Y 446.832,Z 508.578,A -85,B 0,C 180,E1 -8717.859,E2 -8717.859} C_VEL
LIN {X 0,Y 446.461,Z 517.426,A -85,B 0,C 180,E1 -8718.885,E2 -8718.885} C_VEL
LIN {X 0,Y 446.171,Z 524.096,A -85,B 0,C 180,E1 -8719.796,E2 -8719.796} C_VEL
LIN {X 0,Y 445.89,Z 531.066,A -85,B 0,C 180,E1 -8720.934,E2 -8720.934} C_VEL
LIN {X 0,Y 445.698,Z 536.872,A -85,B 0,C 180,E1 -8722.072,E2 -8722.072} C_VEL
LIN {X 0,Y 445.547,Z 541.846,A -85,B 0,C 180,E1 -8723.254,E2 -8723.254} C_VEL
LIN {X 0,Y 445.492,Z 546.253,A -85,B 0,C 180,E1 -8724.571,E2 -8724.571} C_VEL
LIN {X 0,Y 445.426,Z 550.517,A -85,B 0,C 180,E1 -8726.384,E2 -8726.384} C_VEL
LIN {X 0,Y 445.463,Z 552.105,A -85,B 0,C 180,E1 -8727.289,E2 -8727.289} C_VEL
LIN {X 0,Y 445.425,Z 553.713,A -85,B 0,C 180,E1 -8729.098,E2 -8729.098} C_VEL
LIN {X 0,Y 445.403,Z 554.004,A -85,B 0,C 180,E1 -8730.002,E2 -8730.002} C_VEL
LIN {X 0,Y 445.433,Z 553.114,A -85,B 0,C 180,E1 -8731.81,E2 -8731.81} C_VEL
LIN {X 0,Y 445.464,Z 552.096,A -85,B 0,C 180,E1 -8732.714,E2 -8732.714} C_VEL
LIN {X 0,Y 445.431,Z 548.664,A -85,B 0,C 180,E1 -8734.526,E2 -8734.526} C_VEL
LIN {X 0,Y 445.46,Z 545.349,A -85,B 0,C 180,E1 -8735.749,E2 -8735.749} C_VEL
LIN {X 0,Y 445.593,Z 539.912,A -85,B 0,C 180,E1 -8737.25,E2 -8737.25} C_VEL
LIN {X 0,Y 445.769,Z 534.836,A -85,B 0,C 180,E1 -8738.387,E2 -8738.387} C_VEL
LIN {X 0,Y 445.984,Z 528.702,A -85,B 0,C 180,E1 -8739.525,E2 -8739.525} C_VEL
LIN {X 0,Y 446.327,Z 521.285,A -85,B 0,C 180,E1 -8740.663,E2 -8740.663} C_VEL
LIN {X 0,Y 446.816,Z 512.249,A -85,B 0,C 180,E1 -8741.8,E2 -8741.8} C_VEL
LIN {X 0,Y 447.201,Z 503.537,A -85,B 0,C 180,E1 -8742.711,E2 -8742.711} C_VEL
LIN {X 0,Y 447.673,Z 494.094,A -85,B 0,C 180,E1 -8743.526,E2 -8743.526} C_VEL
LIN {X 0,Y 448.089,Z 484.804,A -85,B 0,C 180,E1 -8744.186,E2 -8744.186} C_VEL
LIN {X 0,Y 448.507,Z 474.888,A -85,B 0,C 180,E1 -8744.752,E2 -8744.752} C_VEL
LIN {X 0,Y 448.996,Z 463.838,A -85,B 0,C 180,E1 -8745.229,E2 -8745.229} C_VEL
LIN {X 0,Y 449.243,Z 452.819,A -85,B 0,C 180,E1 -8745.569,E2 -8745.569} C_VEL
LIN {X 0,Y 449.616,Z 433.048,A -85,B 0,C 180,E1 -8745.934,E2 -8745.934} C_VEL
LIN {X 0,Y 450.236,Z 361.44,A -85,B 0,C 180,E1 -8747.173,E2 -8747.173} C_VEL
LIN {X 0,Y 447.951,Z 344.158,A -85,B 0,C 180,E1 -8747.608,E2 -8747.608} C_VEL
LIN {X 0,Y 448.866,Z 323.194,A -85,B 0,C 180,E1 -8750.627,E2 -8750.627} C_VEL
LIN {X 0,Y 449.839,Z 301.9,A -85,B 0,C 180,E1 -8753.722,E2 -8753.722} C_VEL
LIN {X 0,Y 448.46,Z 293.595,A -85,B 0,C 180,E1 -8755.032,E2 -8755.032} C_VEL
LIN {X 0,Y 446.421,Z 284.879,A -85,B 0,C 180,E1 -8756.484,E2 -8756.484} C_VEL
LIN {X 0,Y 446.413,Z 284.885,A -85,B 0,C 180,E1 -8759.211,E2 -8759.211} C_VEL
LIN {X 0,Y 446.413,Z 284.877,A -85,B 0,C 180,E1 -8762.361,E2 -8762.361} C_VEL
LIN {X 0,Y 446.409,Z 284.882,A -85,B 0,C 180,E1 -8765.625,E2 -8765.625} C_VEL
LIN {X 0,Y 446.432,Z 284.877,A -85,B 0,C 180,E1 -8769.026,E2 -8769.026} C_VEL
LIN {X 0,Y 446.423,Z 284.878,A -85,B 0,C 180,E1 -8772.276,E2 -8772.276} C_VEL
LIN {X 0,Y 446.439,Z 284.874,A -85,B 0,C 180,E1 -8775.102,E2 -8775.102} C_VEL
LIN {X 0,Y 446.418,Z 284.876,A -85,B 0,C 180,E1 -8778.608,E2 -8778.608} C_VEL
LIN {X 0,Y 446.451,Z 284.87,A -85,B 0,C 180,E1 -8780.974,E2 -8780.974} C_VEL
LIN {X 0,Y 446.401,Z 284.875,A -85,B 0,C 180,E1 -8784.373,E2 -8784.373} C_VEL
LIN {X 0,Y 446.4,Z 284.871,A -85,B 0,C 180,E1 -8787.637,E2 -8787.637} C_VEL
LIN {X 0,Y 446.445,Z 284.869,A -85,B 0,C 180,E1 -8790.791,E2 -8790.791} C_VEL
LIN {X 0,Y 446.454,Z 284.869,A -85,B 0,C 180,E1 -8793.847,E2 -8793.847} C_VEL
LIN {X 0,Y 446.421,Z 284.878,A -85,B 0,C 180,E1 -8796.823,E2 -8796.823} C_VEL
LIN {X 0,Y 446.432,Z 284.873,A -85,B 0,C 180,E1 -8799.737,E2 -8799.737} C_VEL
LIN {X 0,Y 446.434,Z 284.876,A -85,B 0,C 180,E1 -8802.596,E2 -8802.596} C_VEL
LIN {X 0,Y 446.447,Z 284.872,A -85,B 0,C 180,E1 -8805.412,E2 -8805.412} C_VEL
LIN {X 0,Y 446.517,Z 284.864,A -85,B 0,C 180,E1 -8808.194,E2 -8808.194} C_VEL
LIN {X 0,Y 446.57,Z 284.861,A -85,B 0,C 180,E1 -8811.858,E2 -8811.858} C_VEL
LIN {X 0,Y 446.61,Z 284.859,A -85,B 0,C 180,E1 -8814.583,E2 -8814.583} C_VEL
LIN {X 0,Y 446.746,Z 284.952,A -85,B 0,C 180,E1 -8817.577,E2 -8817.577} C_VEL
LIN {X 0,Y 447.679,Z 288.896,A -85,B 0,C 180,E1 -8818.201,E2 -8818.201} C_VEL
LIN {X 0,Y 447.419,Z 307.527,A -85,B 0,C 180,E1 -8820.901,E2 -8820.901} C_VEL
LIN {X 0,Y 447.143,Z 330.281,A -85,B 0,C 180,E1 -8824.282,E2 -8824.282} C_VEL
LIN {X 0,Y 447.056,Z 337.77,A -85,B 0,C 180,E1 -8825.413,E2 -8825.413} C_VEL
LIN {X 0,Y 449.547,Z 352.551,A -85,B 0,C 180,E1 -8825.833,E2 -8825.833} C_VEL
LIN {X 0,Y 449.792,Z 358.783,A -85,B 0,C 180,E1 -8825.97,E2 -8825.97} C_VEL
LIN {X 0,Y 448.797,Z 421.401,A -85,B 0,C 180,E1 -8827.197,E2 -8827.197} C_VEL
LIN {X 0,Y 448.58,Z 431.997,A -85,B 0,C 180,E1 -8827.54,E2 -8827.54} C_VEL
LIN {X 0,Y 448.203,Z 443.85,A -85,B 0,C 180,E1 -8828.113,E2 -8828.113} C_VEL
LIN {X 0,Y 447.91,Z 453.052,A -85,B 0,C 180,E1 -8828.719,E2 -8828.719} C_VEL
LIN {X 0,Y 447.527,Z 461.134,A -85,B 0,C 180,E1 -8829.377,E2 -8829.377} C_VEL
LIN {X 0,Y 447.121,Z 469.218,A -85,B 0,C 180,E1 -8830.186,E2 -8830.186} C_VEL
LIN {X 0,Y 446.772,Z 476.772,A -85,B 0,C 180,E1 -8831.111,E2 -8831.111} C_VEL
LIN {X 0,Y 446.457,Z 483.77,A -85,B 0,C 180,E1 -8832.162,E2 -8832.162} C_VEL
LIN {X 0,Y 446.092,Z 490.489,A -85,B 0,C 180,E1 -8833.438,E2 -8833.438} C_VEL
LIN {X 0,Y 445.85,Z 495.223,A -85,B 0,C 180,E1 -8834.609,E2 -8834.609} C_VEL
LIN {X 0,Y 445.719,Z 499.156,A -85,B 0,C 180,E1 -8835.894,E2 -8835.894} C_VEL
LIN {X 0,Y 445.621,Z 500.673,A -85,B 0,C 180,E1 -8836.493,E2 -8836.493} C_VEL
LIN {X 0,Y 445.469,Z 502.414,A -85,B 0,C 180,E1 -8837.443,E2 -8837.443} C_VEL
LIN {X 0,Y 445.414,Z 503.971,A -85,B 0,C 180,E1 -8838.8,E2 -8838.8} C_VEL
LIN {X 0,Y 445.37,Z 504.249,A -85,B 0,C 180,E1 -8840.314,E2 -8840.314} C_VEL
LIN {X 0,Y 445.414,Z 503.589,A -85,B 0,C 180,E1 -8841.429,E2 -8841.429} C_VEL
LIN {X 0,Y 445.46,Z 502.638,A -85,B 0,C 180,E1 -8842.25,E2 -8842.25} C_VEL
LIN {X 0,Y 445.612,Z 499.403,A -85,B 0,C 180,E1 -8843.838,E2 -8843.838} C_VEL
LIN {X 0,Y 445.701,Z 496.996,A -85,B 0,C 180,E1 -8844.7,E2 -8844.7} C_VEL
LIN {X 0,Y 445.806,Z 493.757,A -85,B 0,C 180,E1 -8845.625,E2 -8845.625} C_VEL
LIN {X 0,Y 446.038,Z 487.795,A -85,B 0,C 180,E1 -8846.937,E2 -8846.937} C_VEL
LIN {X 0,Y 446.299,Z 482.23,A -85,B 0,C 180,E1 -8847.919,E2 -8847.919} C_VEL
LIN {X 0,Y 446.571,Z 475.132,A -85,B 0,C 180,E1 -8848.943,E2 -8848.943} C_VEL
LIN {X 0,Y 446.902,Z 467.741,A -85,B 0,C 180,E1 -8849.816,E2 -8849.816} C_VEL
LIN {X 0,Y 447.306,Z 458.48,A -85,B 0,C 180,E1 -8850.707,E2 -8850.707} C_VEL
LIN {X 0,Y 447.697,Z 447.235,A -85,B 0,C 180,E1 -8851.531,E2 -8851.531} C_VEL
LIN {X 0,Y 448.007,Z 438.415,A -85,B 0,C 180,E1 -8852.025,E2 -8852.025} C_VEL
LIN {X 0,Y 448.251,Z 428.862,A -85,B 0,C 180,E1 -8852.43,E2 -8852.43} C_VEL
LIN {X 0,Y 448.38,Z 419.057,A -85,B 0,C 180,E1 -8852.719,E2 -8852.719} C_VEL
LIN {X 0,Y 449.049,Z 353.54,A -85,B 0,C 180,E1 -8853.925,E2 -8853.925} C_VEL
LIN {X 0,Y 446.839,Z 339.029,A -85,B 0,C 180,E1 -8854.281,E2 -8854.281} C_VEL
LIN {X 0,Y 447.508,Z 320.994,A -85,B 0,C 180,E1 -8857.77,E2 -8857.77} C_VEL
LIN {X 0,Y 448.121,Z 305.148,A -85,B 0,C 180,E1 -8860.894,E2 -8860.894} C_VEL
LIN {X 0,Y 448.39,Z 295.209,A -85,B 0,C 180,E1 -8862.886,E2 -8862.886} C_VEL
LIN {X 0,Y 446.467,Z 284.873,A -85,B 0,C 180,E1 -8865.102,E2 -8865.102} C_VEL
LIN {X 0,Y 446.42,Z 284.873,A -85,B 0,C 180,E1 -8868.611,E2 -8868.611} C_VEL
LIN {X 0,Y 446.396,Z 284.878,A -85,B 0,C 180,E1 -8871.925,E2 -8871.925} C_VEL
LIN {X 0,Y 446.417,Z 284.876,A -85,B 0,C 180,E1 -8875.478,E2 -8875.478} C_VEL
LIN {X 0,Y 446.407,Z 284.873,A -85,B 0,C 180,E1 -8878.7,E2 -8878.7} C_VEL
LIN {X 0,Y 446.396,Z 284.874,A -85,B 0,C 180,E1 -8878.934,E2 -8878.934} C_VEL
LIN {X 0,Y 445.717,Z 284.965,A -85,B 0,C 180,E1 -8879.688,E2 -8879.688} C_VEL
LIN {X 0,Y 442.848,Z 285.32,A -85,B 0,C 180,E1 -8880.913,E2 -8880.913} C_VEL
LIN {X 0,Y 440.436,Z 285.622,A -85,B 0,C 180,E1 -8881.901,E2 -8881.901} C_VEL
LIN {X 0,Y 439.415,Z 285.747,A -85,B 0,C 180,E1 -8882.664,E2 -8882.664} C_VEL
LIN {X 0,Y 439.339,Z 285.754,A -85,B 0,C 180,E1 -8882.923,E2 -8882.923} C_VEL
LIN {X 0,Y 439.373,Z 285.751,A -85,B 0,C 180,E1 -8885.749,E2 -8885.749} C_VEL
LIN {X 0,Y 439.415,Z 285.752,A -85,B 0,C 180,E1 -8888.416,E2 -8888.416} C_VEL
LIN {X 0,Y 439.426,Z 285.743,A -85,B 0,C 180,E1 -8891.345,E2 -8891.345} C_VEL
LIN {X 0,Y 439.448,Z 285.741,A -85,B 0,C 180,E1 -8894.224,E2 -8894.224} C_VEL
LIN {X 0,Y 439.487,Z 285.735,A -85,B 0,C 180,E1 -8898.001,E2 -8898.001} C_VEL
LIN {X 0,Y 439.485,Z 285.738,A -85,B 0,C 180,E1 -8901.724,E2 -8901.724} C_VEL
LIN {X 0,Y 439.6,Z 285.721,A -85,B 0,C 180,E1 -8904.494,E2 -8904.494} C_VEL
LIN {X 0,Y 439.628,Z 285.719,A -85,B 0,C 180,E1 -8908.166,E2 -8908.166} C_VEL
LIN {X 0,Y 439.672,Z 285.717,A -85,B 0,C 180,E1 -8909.998,E2 -8909.998} C_VEL
LIN {X 0,Y 439.604,Z 285.72,A -85,B 0,C 180,E1 -8912.747,E2 -8912.747} C_VEL
LIN {X 0,Y 439.559,Z 285.73,A -85,B 0,C 180,E1 -8916.424,E2 -8916.424} C_VEL
LIN {X 0,Y 439.478,Z 285.736,A -85,B 0,C 180,E1 -8919.199,E2 -8919.199} C_VEL
LIN {X 0,Y 439.464,Z 285.74,A -85,B 0,C 180,E1 -8922.934,E2 -8922.934} C_VEL
LIN {X 0,Y 439.443,Z 285.745,A -85,B 0,C 180,E1 -8926.344,E2 -8926.344} C_VEL
LIN {X 0,Y 439.396,Z 285.747,A -85,B 0,C 180,E1 -8929.623,E2 -8929.623} C_VEL
LIN {X 0,Y 439.353,Z 285.754,A -85,B 0,C 180,E1 -8932.572,E2 -8932.572} C_VEL
LIN {X 0,Y 439.361,Z 285.754,A -85,B 0,C 180,E1 -8935.583,E2 -8935.583} C_VEL
LIN {X 0,Y 439.383,Z 285.749,A -85,B 0,C 180,E1 -8938.671,E2 -8938.671} C_VEL
LIN {X 0,Y 439.353,Z 285.754,A -85,B 0,C 180,E1 -8942.026,E2 -8942.026} C_VEL
LIN {X 0,Y 439.374,Z 285.752,A -85,B 0,C 180,E1 -8945.336,E2 -8945.336} C_VEL
LIN {X 0,Y 439.347,Z 285.754,A -85,B 0,C 180,E1 -8948.592,E2 -8948.592} C_VEL
LIN {X 0,Y 439.36,Z 285.751,A -85,B 0,C 180,E1 -8951.252,E2 -8951.252} C_VEL
LIN {X 0,Y 439.369,Z 285.753,A -85,B 0,C 180,E1 -8954.725,E2 -8954.725} C_VEL
LIN {X 0,Y 439.363,Z 285.751,A -85,B 0,C 180,E1 -8957.791,E2 -8957.791} C_VEL
LIN {X 0,Y 439.394,Z 285.75,A -85,B 0,C 180,E1 -8960.223,E2 -8960.223} C_VEL
LIN {X 0,Y 439.335,Z 285.754,A -85,B 0,C 180,E1 -8963.708,E2 -8963.708} C_VEL
LIN {X 0,Y 439.329,Z 285.763,A -85,B 0,C 180,E1 -8967.05,E2 -8967.05} C_VEL
LIN {X 0,Y 439.351,Z 285.752,A -85,B 0,C 180,E1 -8970.271,E2 -8970.271} C_VEL
LIN {X 0,Y 439.384,Z 285.757,A -85,B 0,C 180,E1 -8973.393,E2 -8973.393} C_VEL
LIN {X 0,Y 439.338,Z 285.754,A -85,B 0,C 180,E1 -8976.426,E2 -8976.426} C_VEL
LIN {X 0,Y 439.336,Z 285.758,A -85,B 0,C 180,E1 -8979.394,E2 -8979.394} C_VEL
LIN {X 0,Y 439.377,Z 285.752,A -85,B 0,C 180,E1 -8982.307,E2 -8982.307} C_VEL
LIN {X 0,Y 439.395,Z 285.747,A -85,B 0,C 180,E1 -8985.172,E2 -8985.172} C_VEL
LIN {X 0,Y 439.455,Z 285.745,A -85,B 0,C 180,E1 -8988,E2 -8988} C_VEL
LIN {X 0,Y 439.491,Z 285.735,A -85,B 0,C 180,E1 -8991.725,E2 -8991.725} C_VEL
LIN {X 0,Y 439.568,Z 285.733,A -85,B 0,C 180,E1 -8994.495,E2 -8994.495} C_VEL
LIN {X 0,Y 439.579,Z 285.725,A -85,B 0,C 180,E1 -8998.167,E2 -8998.167} C_VEL
LIN {X 0,Y 439.702,Z 285.708,A -85,B 0,C 180,E1 -9000,E2 -9000} C_VEL
LIN {X 0,Y 439.605,Z 285.725,A -85,B 0,C 180,E1 -9002.749,E2 -9002.749} C_VEL
LIN {X 0,Y 439.562,Z 285.726,A -85,B 0,C 180,E1 -9006.426,E2 -9006.426} C_VEL
LIN {X 0,Y 439.442,Z 285.746,A -85,B 0,C 180,E1 -9009.202,E2 -9009.202} C_VEL
LIN {X 0,Y 439.448,Z 285.74,A -85,B 0,C 180,E1 -9012.728,E2 -9012.728} C_VEL
LIN {X 0,Y 439.391,Z 285.749,A -85,B 0,C 180,E1 -9016.35,E2 -9016.35} C_VEL
LIN {X 0,Y 439.351,Z 285.755,A -85,B 0,C 180,E1 -9019.628,E2 -9019.628} C_VEL
LIN {X 0,Y 439.319,Z 285.759,A -85,B 0,C 180,E1 -9022.577,E2 -9022.577} C_VEL
LIN {X 0,Y 439.354,Z 285.752,A -85,B 0,C 180,E1 -9025.588,E2 -9025.588} C_VEL
LIN {X 0,Y 439.368,Z 285.757,A -85,B 0,C 180,E1 -9028.676,E2 -9028.676} C_VEL
LIN {X 0,Y 439.322,Z 285.756,A -85,B 0,C 180,E1 -9032.033,E2 -9032.033} C_VEL
LIN {X 0,Y 439.351,Z 285.755,A -85,B 0,C 180,E1 -9035.344,E2 -9035.344} C_VEL
LIN {X 0,Y 439.334,Z 285.756,A -85,B 0,C 180,E1 -9038.599,E2 -9038.599} C_VEL
LIN {X 0,Y 439.342,Z 285.762,A -85,B 0,C 180,E1 -9041.259,E2 -9041.259} C_VEL
LIN {X 0,Y 439.34,Z 285.754,A -85,B 0,C 180,E1 -9044.736,E2 -9044.736} C_VEL
LIN {X 0,Y 439.362,Z 285.757,A -85,B 0,C 180,E1 -9047.799,E2 -9047.799} C_VEL
LIN {X 0,Y 439.344,Z 285.756,A -85,B 0,C 180,E1 -9050.226,E2 -9050.226} C_VEL
LIN {X 0,Y 439.34,Z 285.758,A -85,B 0,C 180,E1 -9053.716,E2 -9053.716} C_VEL
LIN {X 0,Y 439.346,Z 285.753,A -85,B 0,C 180,E1 -9057.058,E2 -9057.058} C_VEL
LIN {X 0,Y 439.348,Z 285.759,A -85,B 0,C 180,E1 -9060.277,E2 -9060.277} C_VEL
LIN {X 0,Y 439.381,Z 285.825,A -85,B 0,C 180,E1 -9062.821,E2 -9062.821} C_VEL
LIN {X 0,Y 442.904,Z 301.846,A -85,B 0,C 180,E1 -9065.638,E2 -9065.638} C_VEL
LIN {X 0,Y 443.157,Z 304.942,A -85,B 0,C 180,E1 -9066.151,E2 -9066.151} C_VEL
LIN {X 0,Y 441.9,Z 326.439,A -85,B 0,C 180,E1 -9069.524,E2 -9069.524} C_VEL
LIN {X 0,Y 440.835,Z 344.833,A -85,B 0,C 180,E1 -9072.371,E2 -9072.371} C_VEL
LIN {X 0,Y 443.142,Z 364.322,A -85,B 0,C 180,E1 -9072.799,E2 -9072.799} C_VEL
LIN {X 0,Y 442.186,Z 450.198,A -85,B 0,C 180,E1 -9074.298,E2 -9074.298} C_VEL
LIN {X 0,Y 441.933,Z 459.794,A -85,B 0,C 180,E1 -9074.555,E2 -9074.555} C_VEL
LIN {X 0,Y 441.588,Z 470.227,A -85,B 0,C 180,E1 -9074.956,E2 -9074.956} C_VEL
LIN {X 0,Y 441.19,Z 480.325,A -85,B 0,C 180,E1 -9075.473,E2 -9075.473} C_VEL
LIN {X 0,Y 440.767,Z 489.314,A -85,B 0,C 180,E1 -9076.048,E2 -9076.048} C_VEL
LIN {X 0,Y 440.349,Z 499.505,A -85,B 0,C 180,E1 -9076.863,E2 -9076.863} C_VEL
LIN {X 0,Y 439.883,Z 507.842,A -85,B 0,C 180,E1 -9077.664,E2 -9077.664} C_VEL
LIN {X 0,Y 439.446,Z 516.763,A -85,B 0,C 180,E1 -9078.705,E2 -9078.705} C_VEL
LIN {X 0,Y 439.143,Z 523.495,A -85,B 0,C 180,E1 -9079.631,E2 -9079.631} C_VEL
LIN {X 0,Y 438.818,Z 530.513,A -85,B 0,C 180,E1 -9080.787,E2 -9080.787} C_VEL
LIN {X 0,Y 438.573,Z 537.328,A -85,B 0,C 180,E1 -9082.174,E2 -9082.174} C_VEL
LIN {X 0,Y 438.483,Z 541.185,A -85,B 0,C 180,E1 -9083.098,E2 -9083.098} C_VEL
LIN {X 0,Y 438.384,Z 545.788,A -85,B 0,C 180,E1 -9084.483,E2 -9084.483} C_VEL
LIN {X 0,Y 438.353,Z 548.138,A -85,B 0,C 180,E1 -9085.404,E2 -9085.404} C_VEL
LIN {X 0,Y 438.388,Z 551.682,A -85,B 0,C 180,E1 -9087.245,E2 -9087.245} C_VEL
LIN {X 0,Y 438.364,Z 553.31,A -85,B 0,C 180,E1 -9089.083,E2 -9089.083} C_VEL
LIN {X 0,Y 438.341,Z 553.603,A -85,B 0,C 180,E1 -9090.002,E2 -9090.002} C_VEL
LIN {X 0,Y 438.35,Z 552.725,A -85,B 0,C 180,E1 -9091.839,E2 -9091.839} C_VEL
LIN {X 0,Y 438.389,Z 551.708,A -85,B 0,C 180,E1 -9092.758,E2 -9092.758} C_VEL
LIN {X 0,Y 438.358,Z 548.29,A -85,B 0,C 180,E1 -9094.599,E2 -9094.599} C_VEL
LIN {X 0,Y 438.378,Z 544.378,A -85,B 0,C 180,E1 -9096.021,E2 -9096.021} C_VEL
LIN {X 0,Y 438.516,Z 539.559,A -85,B 0,C 180,E1 -9097.368,E2 -9097.368} C_VEL
LIN {X 0,Y 438.697,Z 534.487,A -85,B 0,C 180,E1 -9098.523,E2 -9098.523} C_VEL
LIN {X 0,Y 439.01,Z 526.906,A -85,B 0,C 180,E1 -9099.91,E2 -9099.91} C_VEL
LIN {X 0,Y 439.283,Z 520.932,A -85,B 0,C 180,E1 -9100.836,E2 -9100.836} C_VEL
LIN {X 0,Y 439.827,Z 511.892,A -85,B 0,C 180,E1 -9101.99,E2 -9101.99} C_VEL
LIN {X 0,Y 440.225,Z 503.173,A -85,B 0,C 180,E1 -9102.915,E2 -9102.915} C_VEL
LIN {X 0,Y 440.733,Z 493.873,A -85,B 0,C 180,E1 -9103.731,E2 -9103.731} C_VEL
LIN {X 0,Y 441.173,Z 484.416,A -85,B 0,C 180,E1 -9104.413,E2 -9104.413} C_VEL
LIN {X 0,Y 441.619,Z 474.481,A -85,B 0,C 180,E1 -9104.988,E2 -9104.988} C_VEL
LIN {X 0,Y 442.118,Z 463.438,A -85,B 0,C 180,E1 -9105.472,E2 -9105.472} C_VEL
LIN {X 0,Y 442.414,Z 452.463,A -85,B 0,C 180,E1 -9105.816,E2 -9105.816} C_VEL
LIN {X 0,Y 442.793,Z 432.919,A -85,B 0,C 180,E1 -9106.186,E2 -9106.186} C_VEL
LIN {X 0,Y 443.481,Z 362.082,A -85,B 0,C 180,E1 -9107.442,E2 -9107.442} C_VEL
LIN {X 0,Y 441.061,Z 344.165,A -85,B 0,C 180,E1 -9107.892,E2 -9107.892} C_VEL
LIN {X 0,Y 442.016,Z 323.199,A -85,B 0,C 180,E1 -9110.962,E2 -9110.962} C_VEL
LIN {X 0,Y 443.004,Z 303.509,A -85,B 0,C 180,E1 -9113.862,E2 -9113.862} C_VEL
LIN {X 0,Y 441.738,Z 295.761,A -85,B 0,C 180,E1 -9115.11,E2 -9115.11} C_VEL
LIN {X 0,Y 439.35,Z 285.762,A -85,B 0,C 180,E1 -9116.8,E2 -9116.8} C_VEL
LIN {X 0,Y 439.363,Z 285.762,A -85,B 0,C 180,E1 -9119.726,E2 -9119.726} C_VEL
LIN {X 0,Y 439.364,Z 285.757,A -85,B 0,C 180,E1 -9122.945,E2 -9122.945} C_VEL
LIN {X 0,Y 439.363,Z 285.755,A -85,B 0,C 180,E1 -9126.286,E2 -9126.286} C_VEL
LIN {X 0,Y 439.394,Z 285.756,A -85,B 0,C 180,E1 -9129.849,E2 -9129.849} C_VEL
LIN {X 0,Y 439.372,Z 285.755,A -85,B 0,C 180,E1 -9132.626,E2 -9132.626} C_VEL
LIN {X 0,Y 439.386,Z 285.753,A -85,B 0,C 180,E1 -9135.269,E2 -9135.269} C_VEL
LIN {X 0,Y 439.381,Z 285.752,A -85,B 0,C 180,E1 -9138.741,E2 -9138.741} C_VEL
LIN {X 0,Y 439.371,Z 285.754,A -85,B 0,C 180,E1 -9141.604,E2 -9141.604} C_VEL
LIN {X 0,Y 439.38,Z 285.747,A -85,B 0,C 180,E1 -9144.843,E2 -9144.843} C_VEL
LIN {X 0,Y 439.351,Z 285.754,A -85,B 0,C 180,E1 -9148.138,E2 -9148.138} C_VEL
LIN {X 0,Y 439.402,Z 285.744,A -85,B 0,C 180,E1 -9151.326,E2 -9151.326} C_VEL
LIN {X 0,Y 439.39,Z 285.751,A -85,B 0,C 180,E1 -9154.415,E2 -9154.415} C_VEL
LIN {X 0,Y 439.359,Z 285.754,A -85,B 0,C 180,E1 -9157.425,E2 -9157.425} C_VEL
LIN {X 0,Y 439.414,Z 285.75,A -85,B 0,C 180,E1 -9160.662,E2 -9160.662} C_VEL
LIN {X 0,Y 439.435,Z 285.747,A -85,B 0,C 180,E1 -9164.224,E2 -9164.224} C_VEL
LIN {X 0,Y 439.484,Z 285.739,A -85,B 0,C 180,E1 -9168.002,E2 -9168.002} C_VEL
LIN {X 0,Y 439.519,Z 285.74,A -85,B 0,C 180,E1 -9171.726,E2 -9171.726} C_VEL
LIN {X 0,Y 439.586,Z 285.734,A -85,B 0,C 180,E1 -9174.496,E2 -9174.496} C_VEL
LIN {X 0,Y 439.652,Z 285.93,A -85,B 0,C 180,E1 -9177.309,E2 -9177.309} C_VEL
LIN {X 0,Y 440.9,Z 291.317,A -85,B 0,C 180,E1 -9178.174,E2 -9178.174} C_VEL
LIN {X 0,Y 440.439,Z 313.067,A -85,B 0,C 180,E1 -9181.372,E2 -9181.372} C_VEL
LIN {X 0,Y 440.224,Z 334.314,A -85,B 0,C 180,E1 -9184.579,E2 -9184.579} C_VEL
LIN {X 0,Y 440.193,Z 338.097,A -85,B 0,C 180,E1 -9185.124,E2 -9185.124} C_VEL
LIN {X 0,Y 442.901,Z 354.034,A -85,B 0,C 180,E1 -9185.578,E2 -9185.578} C_VEL
LIN {X 0,Y 442.836,Z 369.3,A -85,B 0,C 180,E1 -9185.893,E2 -9185.893} C_VEL
LIN {X 0,Y 441.968,Z 422.097,A -85,B 0,C 180,E1 -9186.965,E2 -9186.965} C_VEL
LIN {X 0,Y 441.732,Z 433.937,A -85,B 0,C 180,E1 -9187.37,E2 -9187.37} C_VEL
LIN {X 0,Y 441.343,Z 444.226,A -85,B 0,C 180,E1 -9187.895,E2 -9187.895} C_VEL
LIN {X 0,Y 440.981,Z 454.307,A -85,B 0,C 180,E1 -9188.58,E2 -9188.58} C_VEL
LIN {X 0,Y 440.538,Z 462.734,A -85,B 0,C 180,E1 -9189.296,E2 -9189.296} C_VEL
LIN {X 0,Y 440.145,Z 470.609,A -85,B 0,C 180,E1 -9190.117,E2 -9190.117} C_VEL
LIN {X 0,Y 439.686,Z 479.702,A -85,B 0,C 180,E1 -9191.292,E2 -9191.292} C_VEL
LIN {X 0,Y 439.284,Z 486.59,A -85,B 0,C 180,E1 -9192.444,E2 -9192.444} C_VEL
LIN {X 0,Y 439.047,Z 491.372,A -85,B 0,C 180,E1 -9193.422,E2 -9193.422} C_VEL
LIN {X 0,Y 438.844,Z 495.222,A -85,B 0,C 180,E1 -9194.373,E2 -9194.373} C_VEL
LIN {X 0,Y 438.705,Z 498.354,A -85,B 0,C 180,E1 -9195.328,E2 -9195.328} C_VEL
LIN {X 0,Y 438.482,Z 501.759,A -85,B 0,C 180,E1 -9196.769,E2 -9196.769} C_VEL
LIN {X 0,Y 438.36,Z 503.361,A -85,B 0,C 180,E1 -9197.736,E2 -9197.736} C_VEL
LIN {X 0,Y 438.332,Z 504.472,A -85,B 0,C 180,E1 -9198.93,E2 -9198.93} C_VEL
LIN {X 0,Y 438.295,Z 504.699,A -85,B 0,C 180,E1 -9199.678,E2 -9199.678} C_VEL
LIN {X 0,Y 438.304,Z 504.501,A -85,B 0,C 180,E1 -9200.657,E2 -9200.657} C_VEL
LIN {X 0,Y 438.33,Z 503.742,A -85,B 0,C 180,E1 -9201.64,E2 -9201.64} C_VEL
LIN {X 0,Y 438.389,Z 502.401,A -85,B 0,C 180,E1 -9202.629,E2 -9202.629} C_VEL
LIN {X 0,Y 438.536,Z 499.41,A -85,B 0,C 180,E1 -9204.017,E2 -9204.017} C_VEL
LIN {X 0,Y 438.666,Z 496.09,A -85,B 0,C 180,E1 -9205.124,E2 -9205.124} C_VEL
LIN {X 0,Y 438.854,Z 491.674,A -85,B 0,C 180,E1 -9206.266,E2 -9206.266} C_VEL
LIN {X 0,Y 439.067,Z 486.165,A -85,B 0,C 180,E1 -9207.4,E2 -9207.4} C_VEL
LIN {X 0,Y 439.445,Z 478.381,A -85,B 0,C 180,E1 -9208.672,E2 -9208.672} C_VEL
LIN {X 0,Y 439.784,Z 470.324,A -85,B 0,C 180,E1 -9209.697,E2 -9209.697} C_VEL
LIN {X 0,Y 440.177,Z 462.242,A -85,B 0,C 180,E1 -9210.533,E2 -9210.533} C_VEL
LIN {X 0,Y 440.535,Z 453.99,A -85,B 0,C 180,E1 -9211.231,E2 -9211.231} C_VEL
LIN {X 0,Y 440.846,Z 444.897,A -85,B 0,C 180,E1 -9211.85,E2 -9211.85} C_VEL
LIN {X 0,Y 441.188,Z 434.148,A -85,B 0,C 180,E1 -9212.411,E2 -9212.411} C_VEL
LIN {X 0,Y 441.454,Z 421.784,A -85,B 0,C 180,E1 -9212.84,E2 -9212.84} C_VEL
LIN {X 0,Y 441.745,Z 398.989,A -85,B 0,C 180,E1 -9213.291,E2 -9213.291} C_VEL
LIN {X 0,Y 442.214,Z 354.716,A -85,B 0,C 180,E1 -9214.12,E2 -9214.12} C_VEL
LIN {X 0,Y 439.855,Z 339.091,A -85,B 0,C 180,E1 -9214.506,E2 -9214.506} C_VEL
LIN {X 0,Y 440.511,Z 321.756,A -85,B 0,C 180,E1 -9217.897,E2 -9217.897} C_VEL
LIN {X 0,Y 441.189,Z 305.43,A -85,B 0,C 180,E1 -9221.156,E2 -9221.156} C_VEL
LIN {X 0,Y 441.441,Z 296.726,A -85,B 0,C 180,E1 -9222.92,E2 -9222.92} C_VEL
LIN {X 0,Y 439.392,Z 285.754,A -85,B 0,C 180,E1 -9225.326,E2 -9225.326} C_VEL
LIN {X 0,Y 439.38,Z 285.751,A -85,B 0,C 180,E1 -9228.745,E2 -9228.745} C_VEL
LIN {X 0,Y 439.353,Z 285.759,A -85,B 0,C 180,E1 -9231.612,E2 -9231.612} C_VEL
LIN {X 0,Y 439.389,Z 285.747,A -85,B 0,C 180,E1 -9234.845,E2 -9234.845} C_VEL
LIN {X 0,Y 439.367,Z 285.755,A -85,B 0,C 180,E1 -9238.14,E2 -9238.14} C_VEL
LIN {X 0,Y 439.387,Z 285.75,A -85,B 0,C 180,E1 -9241.61,E2 -9241.61} C_VEL
LIN {X 0,Y 439.339,Z 285.754,A -85,B 0,C 180,E1 -9242.923,E2 -9242.923} C_VEL
LIN {X 0,Y 438.688,Z 285.838,A -85,B 0,C 180,E1 -9243.689,E2 -9243.689} C_VEL
LIN {X 0,Y 435.827,Z 286.192,A -85,B 0,C 180,E1 -9244.933,E2 -9244.933} C_VEL
LIN {X 0,Y 433.406,Z 286.496,A -85,B 0,C 180,E1 -9245.938,E2 -9245.938} C_VEL
LIN {X 0,Y 432.38,Z 286.625,A -85,B 0,C 180,E1 -9246.714,E2 -9246.714} C_VEL
LIN {X 0,Y 432.304,Z 286.631,A -85,B 0,C 180,E1 -9246.977,E2 -9246.977} C_VEL
LIN {X 0,Y 432.39,Z 286.627,A -85,B 0,C 180,E1 -9250.516,E2 -9250.516} C_VEL
LIN {X 0,Y 432.425,Z 286.615,A -85,B 0,C 180,E1 -9253.961,E2 -9253.961} C_VEL
LIN {X 0,Y 432.463,Z 286.61,A -85,B 0,C 180,E1 -9257.803,E2 -9257.803} C_VEL
LIN {X 0,Y 432.452,Z 286.615,A -85,B 0,C 180,E1 -9261.588,E2 -9261.588} C_VEL
LIN {X 0,Y 432.556,Z 286.598,A -85,B 0,C 180,E1 -9264.404,E2 -9264.404} C_VEL
LIN {X 0,Y 432.598,Z 286.595,A -85,B 0,C 180,E1 -9268.136,E2 -9268.136} C_VEL
LIN {X 0,Y 432.623,Z 286.595,A -85,B 0,C 180,E1 -9269.998,E2 -9269.998} C_VEL
LIN {X 0,Y 432.558,Z 286.598,A -85,B 0,C 180,E1 -9272.792,E2 -9272.792} C_VEL
LIN {X 0,Y 432.516,Z 286.606,A -85,B 0,C 180,E1 -9276.529,E2 -9276.529} C_VEL
LIN {X 0,Y 432.424,Z 286.615,A -85,B 0,C 180,E1 -9279.351,E2 -9279.351} C_VEL
LIN {X 0,Y 432.43,Z 286.618,A -85,B 0,C 180,E1 -9282.8,E2 -9282.8} C_VEL
LIN {X 0,Y 432.408,Z 286.623,A -85,B 0,C 180,E1 -9286.475,E2 -9286.475} C_VEL
LIN {X 0,Y 432.331,Z 286.626,A -85,B 0,C 180,E1 -9289.957,E2 -9289.957} C_VEL
LIN {X 0,Y 432.307,Z 286.637,A -85,B 0,C 180,E1 -9292.96,E2 -9292.96} C_VEL
LIN {X 0,Y 432.324,Z 286.634,A -85,B 0,C 180,E1 -9294.998,E2 -9294.998} C_VEL
LIN {X 0,Y 432.329,Z 286.627,A -85,B 0,C 180,E1 -9298.122,E2 -9298.122} C_VEL
LIN {X 0,Y 432.304,Z 286.636,A -85,B 0,C 180,E1 -9301.342,E2 -9301.342} C_VEL
LIN {X 0,Y 432.32,Z 286.628,A -85,B 0,C 180,E1 -9304.673,E2 -9304.673} C_VEL
LIN {X 0,Y 432.31,Z 286.634,A -85,B 0,C 180,E1 -9308.146,E2 -9308.146} C_VEL
LIN {X 0,Y 432.303,Z 286.632,A -85,B 0,C 180,E1 -9311.597,E2 -9311.597} C_VEL
LIN {X 0,Y 432.305,Z 286.638,A -85,B 0,C 180,E1 -9314.343,E2 -9314.343} C_VEL
LIN {X 0,Y 432.288,Z 286.633,A -85,B 0,C 180,E1 -9317.011,E2 -9317.011} C_VEL
LIN {X 0,Y 432.301,Z 286.631,A -85,B 0,C 180,E1 -9319.816,E2 -9319.816} C_VEL
LIN {X 0,Y 432.269,Z 286.639,A -85,B 0,C 180,E1 -9323.018,E2 -9323.018} C_VEL
LIN {X 0,Y 432.292,Z 286.631,A -85,B 0,C 180,E1 -9325.998,E2 -9325.998} C_VEL
LIN {X 0,Y 432.35,Z 286.626,A -85,B 0,C 180,E1 -9329.74,E2 -9329.74} C_VEL
LIN {X 0,Y 432.354,Z 286.633,A -85,B 0,C 180,E1 -9333.369,E2 -9333.369} C_VEL
LIN {X 0,Y 432.323,Z 286.63,A -85,B 0,C 180,E1 -9336.02,E2 -9336.02} C_VEL
LIN {X 0,Y 432.299,Z 286.632,A -85,B 0,C 180,E1 -9339.043,E2 -9339.043} C_VEL
LIN {X 0,Y 432.324,Z 286.634,A -85,B 0,C 180,E1 -9342.008,E2 -9342.008} C_VEL
LIN {X 0,Y 432.342,Z 286.625,A -85,B 0,C 180,E1 -9344.924,E2 -9344.924} C_VEL
LIN {X 0,Y 432.428,Z 286.618,A -85,B 0,C 180,E1 -9347.802,E2 -9347.802} C_VEL
LIN {X 0,Y 432.436,Z 286.614,A -85,B 0,C 180,E1 -9351.589,E2 -9351.589} C_VEL
LIN {X 0,Y 432.544,Z 286.606,A -85,B 0,C 180,E1 -9354.405,E2 -9354.405} C_VEL
LIN {X 0,Y 432.549,Z 286.6,A -85,B 0,C 180,E1 -9358.137,E2 -9358.137} C_VEL
LIN {X 0,Y 432.673,Z 286.584,A -85,B 0,C 180,E1 -9359.999,E2 -9359.999} C_VEL
LIN {X 0,Y 432.554,Z 286.604,A -85,B 0,C 180,E1 -9362.793,E2 -9362.793} C_VEL
LIN {X 0,Y 432.516,Z 286.604,A -85,B 0,C 180,E1 -9366.531,E2 -9366.531} C_VEL
LIN {X 0,Y 432.386,Z 286.627,A -85,B 0,C 180,E1 -9369.354,E2 -9369.354} C_VEL
LIN {X 0,Y 432.389,Z 286.619,A -85,B 0,C 180,E1 -9372.812,E2 -9372.812} C_VEL
LIN {X 0,Y 432.357,Z 286.624,A -85,B 0,C 180,E1 -9376.48,E2 -9376.48} C_VEL
LIN {X 0,Y 432.291,Z 286.639,A -85,B 0,C 180,E1 -9379.962,E2 -9379.962} C_VEL
LIN {X 0,Y 432.272,Z 286.634,A -85,B 0,C 180,E1 -9382.966,E2 -9382.966} C_VEL
LIN {X 0,Y 432.314,Z 286.632,A -85,B 0,C 180,E1 -9386.035,E2 -9386.035} C_VEL
LIN {X 0,Y 432.293,Z 286.632,A -85,B 0,C 180,E1 -9389.191,E2 -9389.191} C_VEL
LIN {X 0,Y 432.277,Z 286.638,A -85,B 0,C 180,E1 -9392.446,E2 -9392.446} C_VEL
LIN {X 0,Y 432.301,Z 286.631,A -85,B 0,C 180,E1 -9395.635,E2 -9395.635} C_VEL
LIN {X 0,Y 432.297,Z 286.634,A -85,B 0,C 180,E1 -9398.717,E2 -9398.717} C_VEL
LIN {X 0,Y 432.286,Z 286.634,A -85,B 0,C 180,E1 -9401.802,E2 -9401.802} C_VEL
LIN {X 0,Y 432.297,Z 286.631,A -85,B 0,C 180,E1 -9404.351,E2 -9404.351} C_VEL
LIN {X 0,Y 432.286,Z 286.634,A -85,B 0,C 180,E1 -9407.02,E2 -9407.02} C_VEL
LIN {X 0,Y 432.285,Z 286.64,A -85,B 0,C 180,E1 -9409.828,E2 -9409.828} C_VEL
LIN {X 0,Y 432.27,Z 286.634,A -85,B 0,C 180,E1 -9413.025,E2 -9413.025} C_VEL
LIN {X 0,Y 432.307,Z 286.637,A -85,B 0,C 180,E1 -9416.006,E2 -9416.006} C_VEL
LIN {X 0,Y 432.319,Z 286.629,A -85,B 0,C 180,E1 -9419.495,E2 -9419.495} C_VEL
LIN {X 0,Y 432.345,Z 286.764,A -85,B 0,C 180,E1 -9422.57,E2 -9422.57} C_VEL
LIN {X 0,Y 435.92,Z 302.995,A -85,B 0,C 180,E1 -9425.476,E2 -9425.476} C_VEL
LIN {X 0,Y 436.248,Z 306.097,A -85,B 0,C 180,E1 -9426.002,E2 -9426.002} C_VEL
LIN {X 0,Y 434.995,Z 326.032,A -85,B 0,C 180,E1 -9429.184,E2 -9429.184} C_VEL
LIN {X 0,Y 433.895,Z 344.917,A -85,B 0,C 180,E1 -9432.144,E2 -9432.144} C_VEL
LIN {X 0,Y 436.27,Z 365.299,A -85,B 0,C 180,E1 -9432.599,E2 -9432.599} C_VEL
LIN {X 0,Y 435.26,Z 449.879,A -85,B 0,C 180,E1 -9434.102,E2 -9434.102} C_VEL
LIN {X 0,Y 434.987,Z 459.481,A -85,B 0,C 180,E1 -9434.362,E2 -9434.362} C_VEL
LIN {X 0,Y 434.644,Z 469.921,A -85,B 0,C 180,E1 -9434.77,E2 -9434.77} C_VEL
LIN {X 0,Y 434.257,Z 479.076,A -85,B 0,C 180,E1 -9435.236,E2 -9435.236} C_VEL
LIN {X 0,Y 433.747,Z 489.764,A -85,B 0,C 180,E1 -9435.937,E2 -9435.937} C_VEL
LIN {X 0,Y 433.337,Z 499.496,A -85,B 0,C 180,E1 -9436.735,E2 -9436.735} C_VEL
LIN {X 0,Y 432.837,Z 508.048,A -85,B 0,C 180,E1 -9437.579,E2 -9437.579} C_VEL
LIN {X 0,Y 432.452,Z 516.02,A -85,B 0,C 180,E1 -9438.52,E2 -9438.52} C_VEL
LIN {X 0,Y 432.003,Z 524.255,A -85,B 0,C 180,E1 -9439.694,E2 -9439.694} C_VEL
LIN {X 0,Y 431.712,Z 531.085,A -85,B 0,C 180,E1 -9440.87,E2 -9440.87} C_VEL
LIN {X 0,Y 431.521,Z 536.761,A -85,B 0,C 180,E1 -9442.045,E2 -9442.045} C_VEL
LIN {X 0,Y 431.402,Z 540.636,A -85,B 0,C 180,E1 -9442.985,E2 -9442.985} C_VEL
LIN {X 0,Y 431.286,Z 545.286,A -85,B 0,C 180,E1 -9444.392,E2 -9444.392} C_VEL
LIN {X 0,Y 431.284,Z 547.653,A -85,B 0,C 180,E1 -9445.329,E2 -9445.329} C_VEL
LIN {X 0,Y 431.314,Z 551.24,A -85,B 0,C 180,E1 -9447.2,E2 -9447.2} C_VEL
LIN {X 0,Y 431.274,Z 552.9,A -85,B 0,C 180,E1 -9449.068,E2 -9449.068} C_VEL
LIN {X 0,Y 431.28,Z 553.195,A -85,B 0,C 180,E1 -9450.002,E2 -9450.002} C_VEL
LIN {X 0,Y 431.27,Z 552.349,A -85,B 0,C 180,E1 -9451.869,E2 -9451.869} C_VEL
LIN {X 0,Y 431.315,Z 551.326,A -85,B 0,C 180,E1 -9452.804,E2 -9452.804} C_VEL
LIN {X 0,Y 431.289,Z 547.933,A -85,B 0,C 180,E1 -9454.675,E2 -9454.675} C_VEL
LIN {X 0,Y 431.278,Z 544.495,A -85,B 0,C 180,E1 -9455.979,E2 -9455.979} C_VEL
LIN {X 0,Y 431.429,Z 539.209,A -85,B 0,C 180,E1 -9457.489,E2 -9457.489} C_VEL
LIN {X 0,Y 431.647,Z 534.139,A -85,B 0,C 180,E1 -9458.663,E2 -9458.663} C_VEL
LIN {X 0,Y 431.947,Z 526.553,A -85,B 0,C 180,E1 -9460.074,E2 -9460.074} C_VEL
LIN {X 0,Y 432.268,Z 520.579,A -85,B 0,C 180,E1 -9461.014,E2 -9461.014} C_VEL
LIN {X 0,Y 432.812,Z 511.537,A -85,B 0,C 180,E1 -9462.187,E2 -9462.187} C_VEL
LIN {X 0,Y 433.254,Z 502.849,A -85,B 0,C 180,E1 -9463.127,E2 -9463.127} C_VEL
LIN {X 0,Y 433.791,Z 493.862,A -85,B 0,C 180,E1 -9463.934,E2 -9463.934} C_VEL
LIN {X 0,Y 434.273,Z 484.183,A -85,B 0,C 180,E1 -9464.648,E2 -9464.648} C_VEL
LIN {X 0,Y 434.782,Z 474.323,A -85,B 0,C 180,E1 -9465.229,E2 -9465.229} C_VEL
LIN {X 0,Y 435.299,Z 462.534,A -85,B 0,C 180,E1 -9465.75,E2 -9465.75} C_VEL
LIN {X 0,Y 435.588,Z 452.513,A -85,B 0,C 180,E1 -9466.07,E2 -9466.07} C_VEL
LIN {X 0,Y 435.988,Z 433.111,A -85,B 0,C 180,E1 -9466.446,E2 -9466.446} C_VEL
LIN {X 0,Y 436.775,Z 362.957,A -85,B 0,C 180,E1 -9467.715,E2 -9467.715} C_VEL
LIN {X 0,Y 434.213,Z 344.06,A -85,B 0,C 180,E1 -9468.212,E2 -9468.212} C_VEL
LIN {X 0,Y 435.242,Z 323.28,A -85,B 0,C 180,E1 -9471.304,E2 -9471.304} C_VEL
LIN {X 0,Y 436.184,Z 305.182,A -85,B 0,C 180,E1 -9474.006,E2 -9474.006} C_VEL
LIN {X 0,Y 435.019,Z 297.831,A -85,B 0,C 180,E1 -9475.216,E2 -9475.216} C_VEL
LIN {X 0,Y 432.31,Z 286.643,A -85,B 0,C 180,E1 -9477.142,E2 -9477.142} C_VEL
LIN {X 0,Y 432.338,Z 286.635,A -85,B 0,C 180,E1 -9480.509,E2 -9480.509} C_VEL
LIN {X 0,Y 432.35,Z 286.631,A -85,B 0,C 180,E1 -9484.002,E2 -9484.002} C_VEL
LIN {X 0,Y 432.311,Z 286.636,A -85,B 0,C 180,E1 -9487.196,E2 -9487.196} C_VEL
LIN {X 0,Y 432.324,Z 286.636,A -85,B 0,C 180,E1 -9490.178,E2 -9490.178} C_VEL
LIN {X 0,Y 432.31,Z 286.635,A -85,B 0,C 180,E1 -9493.059,E2 -9493.059} C_VEL
LIN {X 0,Y 432.319,Z 286.634,A -85,B 0,C 180,E1 -9495.664,E2 -9495.664} C_VEL
LIN {X 0,Y 432.35,Z 286.63,A -85,B 0,C 180,E1 -9498.392,E2 -9498.392} C_VEL
LIN {X 0,Y 432.332,Z 286.633,A -85,B 0,C 180,E1 -9501.85,E2 -9501.85} C_VEL
LIN {X 0,Y 432.32,Z 286.626,A -85,B 0,C 180,E1 -9505.322,E2 -9505.322} C_VEL
LIN {X 0,Y 432.301,Z 286.63,A -85,B 0,C 180,E1 -9508.653,E2 -9508.653} C_VEL
LIN {X 0,Y 432.358,Z 286.621,A -85,B 0,C 180,E1 -9511.368,E2 -9511.368} C_VEL
LIN {X 0,Y 432.345,Z 286.628,A -85,B 0,C 180,E1 -9513.967,E2 -9513.967} C_VEL
LIN {X 0,Y 432.308,Z 286.635,A -85,B 0,C 180,E1 -9517.036,E2 -9517.036} C_VEL
LIN {X 0,Y 432.355,Z 286.629,A -85,B 0,C 180,E1 -9520.041,E2 -9520.041} C_VEL
LIN {X 0,Y 432.385,Z 286.624,A -85,B 0,C 180,E1 -9523.521,E2 -9523.521} C_VEL
LIN {X 0,Y 432.417,Z 286.622,A -85,B 0,C 180,E1 -9527.188,E2 -9527.188} C_VEL
LIN {X 0,Y 432.416,Z 286.625,A -85,B 0,C 180,E1 -9530.647,E2 -9530.647} C_VEL
LIN {X 0,Y 432.538,Z 286.612,A -85,B 0,C 180,E1 -9533.47,E2 -9533.47} C_VEL
LIN {X 0,Y 432.368,Z 286.632,A -85,B 0,C 180,E1 -9535.339,E2 -9535.339} C_VEL
LIN {X 0,Y 432.516,Z 286.697,A -85,B 0,C 180,E1 -9536.973,E2 -9536.973} C_VEL
LIN {X 0,Y 434.022,Z 292.311,A -85,B 0,C 180,E1 -9537.913,E2 -9537.913} C_VEL
LIN {X 0,Y 433.704,Z 310.975,A -85,B 0,C 180,E1 -9540.697,E2 -9540.697} C_VEL
LIN {X 0,Y 433.338,Z 333.921,A -85,B 0,C 180,E1 -9544.186,E2 -9544.186} C_VEL
LIN {X 0,Y 433.311,Z 337.979,A -85,B 0,C 180,E1 -9544.798,E2 -9544.798} C_VEL
LIN {X 0,Y 436.242,Z 355.473,A -85,B 0,C 180,E1 -9545.316,E2 -9545.316} C_VEL
LIN {X 0,Y 435.179,Z 421.849,A -85,B 0,C 180,E1 -9546.695,E2 -9546.695} C_VEL
LIN {X 0,Y 434.884,Z 433.2,A -85,B 0,C 180,E1 -9547.079,E2 -9547.079} C_VEL
LIN {X 0,Y 434.484,Z 444.763,A -85,B 0,C 180,E1 -9547.669,E2 -9547.669} C_VEL
LIN {X 0,Y 434.174,Z 453.462,A -85,B 0,C 180,E1 -9548.26,E2 -9548.26} C_VEL
LIN {X 0,Y 433.731,Z 461.917,A -85,B 0,C 180,E1 -9548.972,E2 -9548.972} C_VEL
LIN {X 0,Y 433.228,Z 470.019,A -85,B 0,C 180,E1 -9549.808,E2 -9549.808} C_VEL
LIN {X 0,Y 432.847,Z 477.55,A -85,B 0,C 180,E1 -9550.762,E2 -9550.762} C_VEL
LIN {X 0,Y 432.434,Z 485.229,A -85,B 0,C 180,E1 -9551.96,E2 -9551.96} C_VEL
LIN {X 0,Y 432.061,Z 491.265,A -85,B 0,C 180,E1 -9553.164,E2 -9553.164} C_VEL
LIN {X 0,Y 431.826,Z 495.207,A -85,B 0,C 180,E1 -9554.131,E2 -9554.131} C_VEL
LIN {X 0,Y 431.622,Z 499.677,A -85,B 0,C 180,E1 -9555.585,E2 -9555.585} C_VEL
LIN {X 0,Y 431.366,Z 502.8,A -85,B 0,C 180,E1 -9557.054,E2 -9557.054} C_VEL
LIN {X 0,Y 431.273,Z 504.137,A -85,B 0,C 180,E1 -9558.037,E2 -9558.037} C_VEL
LIN {X 0,Y 431.238,Z 504.932,A -85,B 0,C 180,E1 -9559.06,E2 -9559.06} C_VEL
LIN {X 0,Y 431.203,Z 505.152,A -85,B 0,C 180,E1 -9560.016,E2 -9560.016} C_VEL
LIN {X 0,Y 431.222,Z 504.745,A -85,B 0,C 180,E1 -9561.012,E2 -9561.012} C_VEL
LIN {X 0,Y 431.275,Z 503.717,A -85,B 0,C 180,E1 -9562.013,E2 -9562.013} C_VEL
LIN {X 0,Y 431.418,Z 501.134,A -85,B 0,C 180,E1 -9563.524,E2 -9563.524} C_VEL
LIN {X 0,Y 431.548,Z 498.413,A -85,B 0,C 180,E1 -9564.58,E2 -9564.58} C_VEL
LIN {X 0,Y 431.74,Z 493.155,A -85,B 0,C 180,E1 -9566.073,E2 -9566.073} C_VEL
LIN {X 0,Y 431.931,Z 488.513,A -85,B 0,C 180,E1 -9567.104,E2 -9567.104} C_VEL
LIN {X 0,Y 432.23,Z 482.822,A -85,B 0,C 180,E1 -9568.135,E2 -9568.135} C_VEL
LIN {X 0,Y 432.522,Z 475.811,A -85,B 0,C 180,E1 -9569.175,E2 -9569.175} C_VEL
LIN {X 0,Y 432.882,Z 468.321,A -85,B 0,C 180,E1 -9570.084,E2 -9570.084} C_VEL
LIN {X 0,Y 433.284,Z 459.787,A -85,B 0,C 180,E1 -9570.932,E2 -9570.932} C_VEL
LIN {X 0,Y 433.713,Z 448.931,A -85,B 0,C 180,E1 -9571.779,E2 -9571.779} C_VEL
LIN {X 0,Y 434.088,Z 438.773,A -85,B 0,C 180,E1 -9572.371,E2 -9572.371} C_VEL
LIN {X 0,Y 434.339,Z 429.277,A -85,B 0,C 180,E1 -9572.785,E2 -9572.785} C_VEL
LIN {X 0,Y 434.494,Z 420.274,A -85,B 0,C 180,E1 -9573.064,E2 -9573.064} C_VEL
LIN {X 0,Y 435.28,Z 355.207,A -85,B 0,C 180,E1 -9574.325,E2 -9574.325} C_VEL
LIN {X 0,Y 432.855,Z 339.122,A -85,B 0,C 180,E1 -9574.737,E2 -9574.737} C_VEL
LIN {X 0,Y 433.531,Z 322.516,A -85,B 0,C 180,E1 -9578.027,E2 -9578.027} C_VEL
LIN {X 0,Y 434.24,Z 306.499,A -85,B 0,C 180,E1 -9581.264,E2 -9581.264} C_VEL
LIN {X 0,Y 434.465,Z 297.866,A -85,B 0,C 180,E1 -9583.037,E2 -9583.037} C_VEL
LIN {X 0,Y 432.355,Z 286.631,A -85,B 0,C 180,E1 -9585.536,E2 -9585.536} C_VEL
LIN {X 0,Y 432.324,Z 286.629,A -85,B 0,C 180,E1 -9588.4,E2 -9588.4} C_VEL
LIN {X 0,Y 432.319,Z 286.632,A -85,B 0,C 180,E1 -9591.85,E2 -9591.85} C_VEL
LIN {X 0,Y 432.323,Z 286.63,A -85,B 0,C 180,E1 -9595.323,E2 -9595.323} C_VEL
LIN {X 0,Y 432.315,Z 286.629,A -85,B 0,C 180,E1 -9598.655,E2 -9598.655} C_VEL
LIN {X 0,Y 432.32,Z 286.633,A -85,B 0,C 180,E1 -9601.873,E2 -9601.873} C_VEL
LIN {X 0,Y 432.324,Z 286.628,A -85,B 0,C 180,E1 -9604.998,E2 -9604.998} C_VEL
LIN {X 0,Y 432.304,Z 286.631,A -85,B 0,C 180,E1 -9606.977,E2 -9606.977} C_VEL
LIN {X 0,Y 431.67,Z 286.714,A -85,B 0,C 180,E1 -9607.755,E2 -9607.755} C_VEL
LIN {X 0,Y 428.868,Z 287.068,A -85,B 0,C 180,E1 -9609.02,E2 -9609.02} C_VEL
LIN {X 0,Y 426.472,Z 287.366,A -85,B 0,C 180,E1 -9610.041,E2 -9610.041} C_VEL
LIN {X 0,Y 425.426,Z 287.492,A -85,B 0,C 180,E1 -9610.829,E2 -9610.829} C_VEL
LIN {X 0,Y 425.333,Z 287.501,A -85,B 0,C 180,E1 -9611.096,E2 -9611.096} C_VEL
LIN {X 0,Y 425.388,Z 287.491,A -85,B 0,C 180,E1 -9613.688,E2 -9613.688} C_VEL
LIN {X 0,Y 425.417,Z 287.489,A -85,B 0,C 180,E1 -9617.598,E2 -9617.598} C_VEL
LIN {X 0,Y 425.4,Z 287.496,A -85,B 0,C 180,E1 -9621.448,E2 -9621.448} C_VEL
LIN {X 0,Y 425.514,Z 287.476,A -85,B 0,C 180,E1 -9624.311,E2 -9624.311} C_VEL
LIN {X 0,Y 425.567,Z 287.471,A -85,B 0,C 180,E1 -9628.106,E2 -9628.106} C_VEL
LIN {X 0,Y 425.576,Z 287.473,A -85,B 0,C 180,E1 -9629.998,E2 -9629.998} C_VEL
LIN {X 0,Y 425.513,Z 287.476,A -85,B 0,C 180,E1 -9632.838,E2 -9632.838} C_VEL
LIN {X 0,Y 425.511,Z 287.48,A -85,B 0,C 180,E1 -9635.685,E2 -9635.685} C_VEL
LIN {X 0,Y 425.396,Z 287.494,A -85,B 0,C 180,E1 -9638.548,E2 -9638.548} C_VEL
LIN {X 0,Y 425.411,Z 287.497,A -85,B 0,C 180,E1 -9642.399,E2 -9642.399} C_VEL
LIN {X 0,Y 425.384,Z 287.495,A -85,B 0,C 180,E1 -9646.308,E2 -9646.308} C_VEL
LIN {X 0,Y 425.322,Z 287.5,A -85,B 0,C 180,E1 -9649.631,E2 -9649.631} C_VEL
LIN {X 0,Y 425.28,Z 287.506,A -85,B 0,C 180,E1 -9652.335,E2 -9652.335} C_VEL
LIN {X 0,Y 425.307,Z 287.504,A -85,B 0,C 180,E1 -9654.652,E2 -9654.652} C_VEL
LIN {X 0,Y 425.256,Z 287.513,A -85,B 0,C 180,E1 -9657.559,E2 -9657.559} C_VEL
LIN {X 0,Y 425.275,Z 287.506,A -85,B 0,C 180,E1 -9660.756,E2 -9660.756} C_VEL
LIN {X 0,Y 425.292,Z 287.505,A -85,B 0,C 180,E1 -9664.283,E2 -9664.283} C_VEL
LIN {X 0,Y 425.255,Z 287.514,A -85,B 0,C 180,E1 -9667.69,E2 -9667.69} C_VEL
LIN {X 0,Y 425.253,Z 287.511,A -85,B 0,C 180,E1 -9670.515,E2 -9670.515} C_VEL
LIN {X 0,Y 425.228,Z 287.511,A -85,B 0,C 180,E1 -9673.346,E2 -9673.346} C_VEL
LIN {X 0,Y 425.227,Z 287.517,A -85,B 0,C 180,E1 -9676.645,E2 -9676.645} C_VEL
LIN {X 0,Y 425.254,Z 287.509,A -85,B 0,C 180,E1 -9679.868,E2 -9679.868} C_VEL
LIN {X 0,Y 425.241,Z 287.515,A -85,B 0,C 180,E1 -9682.484,E2 -9682.484} C_VEL
LIN {X 0,Y 425.246,Z 287.509,A -85,B 0,C 180,E1 -9685.811,E2 -9685.811} C_VEL
LIN {X 0,Y 425.256,Z 287.515,A -85,B 0,C 180,E1 -9689.234,E2 -9689.234} C_VEL
LIN {X 0,Y 425.305,Z 287.502,A -85,B 0,C 180,E1 -9692.439,E2 -9692.439} C_VEL
LIN {X 0,Y 425.304,Z 287.509,A -85,B 0,C 180,E1 -9695.599,E2 -9695.599} C_VEL
LIN {X 0,Y 425.242,Z 287.509,A -85,B 0,C 180,E1 -9698.678,E2 -9698.678} C_VEL
LIN {X 0,Y 425.28,Z 287.511,A -85,B 0,C 180,E1 -9701.7,E2 -9701.7} C_VEL
LIN {X 0,Y 425.295,Z 287.504,A -85,B 0,C 180,E1 -9704.668,E2 -9704.668} C_VEL
LIN {X 0,Y 425.377,Z 287.494,A -85,B 0,C 180,E1 -9707.597,E2 -9707.597} C_VEL
LIN {X 0,Y 425.387,Z 287.491,A -85,B 0,C 180,E1 -9711.448,E2 -9711.448} C_VEL
LIN {X 0,Y 425.501,Z 287.482,A -85,B 0,C 180,E1 -9714.312,E2 -9714.312} C_VEL
LIN {X 0,Y 425.519,Z 287.476,A -85,B 0,C 180,E1 -9718.107,E2 -9718.107} C_VEL
LIN {X 0,Y 425.643,Z 287.46,A -85,B 0,C 180,E1 -9719.999,E2 -9719.999} C_VEL
LIN {X 0,Y 425.506,Z 287.482,A -85,B 0,C 180,E1 -9722.84,E2 -9722.84} C_VEL
LIN {X 0,Y 425.474,Z 287.482,A -85,B 0,C 180,E1 -9726.639,E2 -9726.639} C_VEL
LIN {X 0,Y 425.345,Z 287.504,A -85,B 0,C 180,E1 -9729.51,E2 -9729.51} C_VEL
LIN {X 0,Y 425.349,Z 287.497,A -85,B 0,C 180,E1 -9732.911,E2 -9732.911} C_VEL
LIN {X 0,Y 425.306,Z 287.502,A -85,B 0,C 180,E1 -9736.606,E2 -9736.606} C_VEL
LIN {X 0,Y 425.276,Z 287.509,A -85,B 0,C 180,E1 -9739.637,E2 -9739.637} C_VEL
LIN {X 0,Y 425.24,Z 287.516,A -85,B 0,C 180,E1 -9742.341,E2 -9742.341} C_VEL
LIN {X 0,Y 425.245,Z 287.509,A -85,B 0,C 180,E1 -9745.448,E2 -9745.448} C_VEL
LIN {X 0,Y 425.282,Z 287.512,A -85,B 0,C 180,E1 -9748.635,E2 -9748.635} C_VEL
LIN {X 0,Y 425.218,Z 287.513,A -85,B 0,C 180,E1 -9751.93,E2 -9751.93} C_VEL
LIN {X 0,Y 425.256,Z 287.511,A -85,B 0,C 180,E1 -9755.339,E2 -9755.339} C_VEL
LIN {X 0,Y 425.256,Z 287.513,A -85,B 0,C 180,E1 -9758.903,E2 -9758.903} C_VEL
LIN {X 0,Y 425.244,Z 287.51,A -85,B 0,C 180,E1 -9761.961,E2 -9761.961} C_VEL
LIN {X 0,Y 425.249,Z 287.514,A -85,B 0,C 180,E1 -9765.287,E2 -9765.287} C_VEL
LIN {X 0,Y 425.239,Z 287.51,A -85,B 0,C 180,E1 -9768.625,E2 -9768.625} C_VEL
LIN {X 0,Y 425.251,Z 287.509,A -85,B 0,C 180,E1 -9771.103,E2 -9771.103} C_VEL
LIN {X 0,Y 425.267,Z 287.508,A -85,B 0,C 180,E1 -9774.667,E2 -9774.667} C_VEL
LIN {X 0,Y 425.239,Z 287.517,A -85,B 0,C 180,E1 -9778.077,E2 -9778.077} C_VEL
LIN {X 0,Y 425.275,Z 287.51,A -85,B 0,C 180,E1 -9781.369,E2 -9781.369} C_VEL
LIN {X 0,Y 425.309,Z 287.675,A -85,B 0,C 180,E1 -9782.311,E2 -9782.311} C_VEL
LIN {X 0,Y 429.26,Z 305.699,A -85,B 0,C 180,E1 -9785.586,E2 -9785.586} C_VEL
LIN {X 0,Y 428.833,Z 314.912,A -85,B 0,C 180,E1 -9787.098,E2 -9787.098} C_VEL
LIN {X 0,Y 427.452,Z 336.358,A -85,B 0,C 180,E1 -9790.557,E2 -9790.557} C_VEL
LIN {X 0,Y 426.962,Z 344.664,A -85,B 0,C 180,E1 -9791.884,E2 -9791.884} C_VEL
LIN {X 0,Y 429.397,Z 365.968,A -85,B 0,C 180,E1 -9792.386,E2 -9792.386} C_VEL
LIN {X 0,Y 428.341,Z 449.55,A -85,B 0,C 180,E1 -9793.899,E2 -9793.899} C_VEL
LIN {X 0,Y 428.039,Z 459.166,A -85,B 0,C 180,E1 -9794.163,E2 -9794.163} C_VEL
LIN {X 0,Y 427.692,Z 469.612,A -85,B 0,C 180,E1 -9794.577,E2 -9794.577} C_VEL
LIN {X 0,Y 427.242,Z 479.708,A -85,B 0,C 180,E1 -9795.11,E2 -9795.11} C_VEL
LIN {X 0,Y 426.779,Z 488.696,A -85,B 0,C 180,E1 -9795.703,E2 -9795.703} C_VEL
LIN {X 0,Y 426.321,Z 499.062,A -85,B 0,C 180,E1 -9796.561,E2 -9796.561} C_VEL
LIN {X 0,Y 425.792,Z 508.254,A -85,B 0,C 180,E1 -9797.492,E2 -9797.492} C_VEL
LIN {X 0,Y 425.469,Z 515.278,A -85,B 0,C 180,E1 -9798.329,E2 -9798.329} C_VEL
LIN {X 0,Y 424.968,Z 523.577,A -85,B 0,C 180,E1 -9799.522,E2 -9799.522} C_VEL
LIN {X 0,Y 424.668,Z 530.465,A -85,B 0,C 180,E1 -9800.717,E2 -9800.717} C_VEL
LIN {X 0,Y 424.476,Z 536.191,A -85,B 0,C 180,E1 -9801.912,E2 -9801.912} C_VEL
LIN {X 0,Y 424.291,Z 541.705,A -85,B 0,C 180,E1 -9803.344,E2 -9803.344} C_VEL
LIN {X 0,Y 424.241,Z 545.993,A -85,B 0,C 180,E1 -9804.775,E2 -9804.775} C_VEL
LIN {X 0,Y 424.142,Z 549.164,A -85,B 0,C 180,E1 -9806.202,E2 -9806.202} C_VEL
LIN {X 0,Y 424.242,Z 550.792,A -85,B 0,C 180,E1 -9807.154,E2 -9807.154} C_VEL
LIN {X 0,Y 424.188,Z 552.489,A -85,B 0,C 180,E1 -9809.053,E2 -9809.053} C_VEL
LIN {X 0,Y 424.204,Z 552.785,A -85,B 0,C 180,E1 -9810.002,E2 -9810.002} C_VEL
LIN {X 0,Y 424.193,Z 551.972,A -85,B 0,C 180,E1 -9811.901,E2 -9811.901} C_VEL
LIN {X 0,Y 424.224,Z 550.944,A -85,B 0,C 180,E1 -9812.85,E2 -9812.85} C_VEL
LIN {X 0,Y 424.218,Z 547.575,A -85,B 0,C 180,E1 -9814.753,E2 -9814.753} C_VEL
LIN {X 0,Y 424.239,Z 543.414,A -85,B 0,C 180,E1 -9816.301,E2 -9816.301} C_VEL
LIN {X 0,Y 424.355,Z 538.856,A -85,B 0,C 180,E1 -9817.615,E2 -9817.615} C_VEL
LIN {X 0,Y 424.591,Z 533.804,A -85,B 0,C 180,E1 -9818.808,E2 -9818.808} C_VEL
LIN {X 0,Y 424.913,Z 526.243,A -85,B 0,C 180,E1 -9820.243,E2 -9820.243} C_VEL
LIN {X 0,Y 425.348,Z 518.567,A -85,B 0,C 180,E1 -9821.437,E2 -9821.437} C_VEL
LIN {X 0,Y 425.78,Z 511.29,A -85,B 0,C 180,E1 -9822.392,E2 -9822.392} C_VEL
LIN {X 0,Y 426.316,Z 502.619,A -85,B 0,C 180,E1 -9823.345,E2 -9823.345} C_VEL
LIN {X 0,Y 426.88,Z 493.651,A -85,B 0,C 180,E1 -9824.164,E2 -9824.164} C_VEL
LIN {X 0,Y 427.41,Z 484,A -85,B 0,C 180,E1 -9824.888,E2 -9824.888} C_VEL
LIN {X 0,Y 428.007,Z 472.971,A -85,B 0,C 180,E1 -9825.537,E2 -9825.537} C_VEL
LIN {X 0,Y 428.485,Z 462.454,A -85,B 0,C 180,E1 -9826.008,E2 -9826.008} C_VEL
LIN {X 0,Y 428.774,Z 452.564,A -85,B 0,C 180,E1 -9826.333,E2 -9826.333} C_VEL
LIN {X 0,Y 429.204,Z 433.402,A -85,B 0,C 180,E1 -9826.713,E2 -9826.713} C_VEL
LIN {X 0,Y 430.02,Z 363.363,A -85,B 0,C 180,E1 -9828.016,E2 -9828.016} C_VEL
LIN {X 0,Y 427.354,Z 344.053,A -85,B 0,C 180,E1 -9828.532,E2 -9828.532} C_VEL
LIN {X 0,Y 428.44,Z 323.32,A -85,B 0,C 180,E1 -9831.659,E2 -9831.659} C_VEL
LIN {X 0,Y 429.394,Z 306.957,A -85,B 0,C 180,E1 -9834.153,E2 -9834.153} C_VEL
LIN {X 0,Y 428.111,Z 299.125,A -85,B 0,C 180,E1 -9835.46,E2 -9835.46} C_VEL
LIN {X 0,Y 425.269,Z 287.52,A -85,B 0,C 180,E1 -9837.562,E2 -9837.562} C_VEL
LIN {X 0,Y 425.28,Z 287.514,A -85,B 0,C 180,E1 -9840.815,E2 -9840.815} C_VEL
LIN {X 0,Y 425.302,Z 287.508,A -85,B 0,C 180,E1 -9844.287,E2 -9844.287} C_VEL
LIN {X 0,Y 425.268,Z 287.516,A -85,B 0,C 180,E1 -9847.693,E2 -9847.693} C_VEL
LIN {X 0,Y 425.269,Z 287.513,A -85,B 0,C 180,E1 -9850.519,E2 -9850.519} C_VEL
LIN {X 0,Y 425.25,Z 287.517,A -85,B 0,C 180,E1 -9853.35,E2 -9853.35} C_VEL
LIN {X 0,Y 425.242,Z 287.514,A -85,B 0,C 180,E1 -9856.648,E2 -9856.648} C_VEL
LIN {X 0,Y 425.281,Z 287.51,A -85,B 0,C 180,E1 -9859.476,E2 -9859.476} C_VEL
LIN {X 0,Y 425.268,Z 287.508,A -85,B 0,C 180,E1 -9862.486,E2 -9862.486} C_VEL
LIN {X 0,Y 425.287,Z 287.505,A -85,B 0,C 180,E1 -9865.816,E2 -9865.816} C_VEL
LIN {X 0,Y 425.277,Z 287.502,A -85,B 0,C 180,E1 -9869.236,E2 -9869.236} C_VEL
LIN {X 0,Y 425.327,Z 287.502,A -85,B 0,C 180,E1 -9872.441,E2 -9872.441} C_VEL
LIN {X 0,Y 425.333,Z 287.501,A -85,B 0,C 180,E1 -9875.602,E2 -9875.602} C_VEL
LIN {X 0,Y 425.294,Z 287.509,A -85,B 0,C 180,E1 -9878.682,E2 -9878.682} C_VEL
LIN {X 0,Y 425.305,Z 287.506,A -85,B 0,C 180,E1 -9881.702,E2 -9881.702} C_VEL
LIN {X 0,Y 425.322,Z 287.506,A -85,B 0,C 180,E1 -9884.67,E2 -9884.67} C_VEL
LIN {X 0,Y 425.404,Z 287.494,A -85,B 0,C 180,E1 -9887.598,E2 -9887.598} C_VEL
LIN {X 0,Y 425.414,Z 287.498,A -85,B 0,C 180,E1 -9891.45,E2 -9891.45} C_VEL
LIN {X 0,Y 425.52,Z 287.486,A -85,B 0,C 180,E1 -9894.313,E2 -9894.313} C_VEL
LIN {X 0,Y 425.384,Z 287.52,A -85,B 0,C 180,E1 -9896.626,E2 -9896.626} C_VEL
LIN {X 0,Y 427.29,Z 294.927,A -85,B 0,C 180,E1 -9897.88,E2 -9897.88} C_VEL
LIN {X 0,Y 426.805,Z 313.587,A -85,B 0,C 180,E1 -9900.708,E2 -9900.708} C_VEL
LIN {X 0,Y 426.474,Z 335.085,A -85,B 0,C 180,E1 -9904.017,E2 -9904.017} C_VEL
LIN {X 0,Y 426.454,Z 338.206,A -85,B 0,C 180,E1 -9904.461,E2 -9904.461} C_VEL
LIN {X 0,Y 429.391,Z 355.312,A -85,B 0,C 180,E1 -9904.989,E2 -9904.989} C_VEL
LIN {X 0,Y 429.62,Z 359.915,A -85,B 0,C 180,E1 -9905.104,E2 -9905.104} C_VEL
LIN {X 0,Y 428.401,Z 421.585,A -85,B 0,C 180,E1 -9906.417,E2 -9906.417} C_VEL
LIN {X 0,Y 428.081,Z 431.611,A -85,B 0,C 180,E1 -9906.748,E2 -9906.748} C_VEL
LIN {X 0,Y 427.724,Z 443.395,A -85,B 0,C 180,E1 -9907.317,E2 -9907.317} C_VEL
LIN {X 0,Y 427.306,Z 453.959,A -85,B 0,C 180,E1 -9908.037,E2 -9908.037} C_VEL
LIN {X 0,Y 426.882,Z 461.591,A -85,B 0,C 180,E1 -9908.682,E2 -9908.682} C_VEL
LIN {X 0,Y 426.308,Z 470.485,A -85,B 0,C 180,E1 -9909.609,E2 -9909.609} C_VEL
LIN {X 0,Y 425.953,Z 477.134,A -85,B 0,C 180,E1 -9910.457,E2 -9910.457} C_VEL
LIN {X 0,Y 425.556,Z 483.502,A -85,B 0,C 180,E1 -9911.431,E2 -9911.431} C_VEL
LIN {X 0,Y 425.194,Z 488.806,A -85,B 0,C 180,E1 -9912.409,E2 -9912.409} C_VEL
LIN {X 0,Y 424.924,Z 493.208,A -85,B 0,C 180,E1 -9913.389,E2 -9913.389} C_VEL
LIN {X 0,Y 424.723,Z 496.843,A -85,B 0,C 180,E1 -9914.372,E2 -9914.372} C_VEL
LIN {X 0,Y 424.509,Z 500.826,A -85,B 0,C 180,E1 -9915.779,E2 -9915.779} C_VEL
LIN {X 0,Y 424.416,Z 502.15,A -85,B 0,C 180,E1 -9916.351,E2 -9916.351} C_VEL
LIN {X 0,Y 424.266,Z 503.847,A -85,B 0,C 180,E1 -9917.348,E2 -9917.348} C_VEL
LIN {X 0,Y 424.17,Z 504.916,A -85,B 0,C 180,E1 -9918.35,E2 -9918.35} C_VEL
LIN {X 0,Y 424.128,Z 505.436,A -85,B 0,C 180,E1 -9919.355,E2 -9919.355} C_VEL
LIN {X 0,Y 424.115,Z 505.408,A -85,B 0,C 180,E1 -9920.365,E2 -9920.365} C_VEL
LIN {X 0,Y 424.172,Z 504.232,A -85,B 0,C 180,E1 -9921.907,E2 -9921.907} C_VEL
LIN {X 0,Y 424.307,Z 501.782,A -85,B 0,C 180,E1 -9923.424,E2 -9923.424} C_VEL
LIN {X 0,Y 424.499,Z 497.699,A -85,B 0,C 180,E1 -9924.973,E2 -9924.973} C_VEL
LIN {X 0,Y 424.709,Z 492.97,A -85,B 0,C 180,E1 -9926.274,E2 -9926.274} C_VEL
LIN {X 0,Y 424.985,Z 486.851,A -85,B 0,C 180,E1 -9927.584,E2 -9927.584} C_VEL
LIN {X 0,Y 425.358,Z 479.171,A -85,B 0,C 180,E1 -9928.879,E2 -9928.879} C_VEL
LIN {X 0,Y 425.757,Z 470.95,A -85,B 0,C 180,E1 -9929.957,E2 -9929.957} C_VEL
